(* Logix 5000 project; controller reports 1756-L63 rev 20.15; software revision 20.04; part 35 of 52 *)

        [32].log_data[44].total := -1012.85846, [32].log_data[44].time := 3600.0, [32].log_data[44].valid := 1, [32].log_data[45].time := 3600.0, [32].log_data[45].valid := 1, [32].log_data[46].time := 3600.0, [32].log_data[46].valid := 1, [32].log_data[47].time := 3600.0, [32].log_data[47].valid := 1, [32].log_data[48].min := 6.578031, [32].log_data[48].max := 6.9292355, [32].log_data[48].total := 24261.766, [32].log_data[48].time := 3600.0, [32].log_data[48].minminute := 9, [32].log_data[48].maxminute := 51, [32].log_data[48].valid := 1, [32].log_data[49].min := 7.0189543, [32].log_data[49].max := 9.474559, [32].log_data[49].total := 29951.562, [32].log_data[49].time := 3600.0, [32].log_data[49].minminute := 8, [32].log_data[49].maxminute := 45, [32].log_data[49].valid := 1, [32].log_data[50].min := 2.0610397, [32].log_data[50].max := 2.1768122, [32].log_data[50].total := 7588.2583, [32].log_data[50].time := 3600.0, [32].log_data[50].minminute := 44, [32].log_data[50].maxminute := 52, [32].log_data[50].valid := 1, [32].log_data[51].time := 3600.0, [32].log_data[51].valid := 1, [32].log_data[52].min := -3.0, [32].log_data[52].max := 0.13999939, [32].log_data[52].total := -7599.1304, [32].log_data[52].time := 3600.0, [32].log_data[52].minminute := 11, [32].log_data[52].valid := 1, [32].log_data[53].min := -2.5200043, [32].log_data[53].max := 0.17999268, [32].log_data[53].total := -6900.277, [32].log_data[53].time := 3600.0, [32].log_data[53].minminute := 27, [32].log_data[53].maxminute := 16, [32].log_data[53].valid := 1, [32].log_data[54].max := 0.554, [32].log_data[54].total := 1229.82, [32].log_data[54].time := 3600.0, [32].log_data[54].maxminute := 11, [32].log_data[54].valid := 1, [32].log_data[55].max := 0.523, [32].log_data[55].total := 1217.2505, [32].log_data[55].time := 3600.0, [32].log_data[55].minminute := 4, [32].log_data[55].maxminute := 58, [32].log_data[55].valid := 1, [32].log_data[56].min := 0.16024561, [32].log_data[56].max := 0.16067745, [32].log_data[56].total := 577.5993, [32].log_data[56].time := 3600.0,
        [32].log_data[56].minminute := 58, [32].log_data[56].maxminute := 2, [32].log_data[56].valid := 1, [32].log_data[57].min := 0.29596147, [32].log_data[57].max := 0.2979244, [32].log_data[57].total := 1067.1407, [32].log_data[57].time := 3600.0, [32].log_data[57].minminute := 25, [32].log_data[57].maxminute := 3, [32].log_data[57].valid := 1, [32].log_data[58].time := 3600.0, [32].log_data[58].valid := 1, [32].log_data[59].time := 3600.0, [32].log_data[59].valid := 1, [32].log_data[60].valid := 1, [32].log_data[61].valid := 1, [32].log_data[62].valid := 1, [32].log_data[63].valid := 1, [32].log_data[64].valid := 1, [32].log_data[65].valid := 1, [32].log_data[66].valid := 1, [32].log_data[67].valid := 1, [32].log_data[68].valid := 1, [32].log_data[69].valid := 1, [32].log_data[70].valid := 1, [32].log_data[71].valid := 1, [32].log_data[72].valid := 1, [32].log_data[73].valid := 1, [32].log_data[74].valid := 1, [32].log_data[75].valid := 1, [32].log_data[76].valid := 1, [32].log_data[77].valid := 1, [32].log_data[78].valid := 1, [32].log_data[79].valid := 1, [32].log_data[80].valid := 1, [32].log_data[81].valid := 1, [32].log_data[82].valid := 1, [32].log_data[83].valid := 1, [32].log_data[84].valid := 1, [32].log_data[85].valid := 1, [32].log_data[86].valid := 1, [32].log_data[87].valid := 1, [32].log_data[88].valid := 1, [32].log_data[89].valid := 1, [32].log_data[90].valid := 1, [32].log_data[91].valid := 1, [32].log_data[92].valid := 1, [32].log_data[93].valid := 1, [32].log_data[94].valid := 1, [32].log_data[95].valid := 1, [32].log_data[96].valid := 1, [32].log_data[97].valid := 1, [32].log_data[98].valid := 1, [32].log_data[99].valid := 1, [32].log_data[100].valid := 1, [32].log_data[101].valid := 1, [32].log_data[102].valid := 1, [32].log_data[103].valid := 1, [32].log_data[104].valid := 1, [32].log_data[105].valid := 1,
        [32].log_data[106].valid := 1, [32].log_data[107].valid := 1, [32].log_data[108].valid := 1, [32].log_data[109].valid := 1, [32].log_data[110].valid := 1, [32].log_data[111].valid := 1, [32].log_data[112].valid := 1, [32].log_data[113].valid := 1, [32].log_data[114].valid := 1, [32].log_data[115].valid := 1, [32].log_data[116].valid := 1, [32].log_data[117].valid := 1, [32].log_data[118].valid := 1, [32].log_data[119].valid := 1, [32].log_data[120].valid := 1, [32].log_data[121].valid := 1, [32].log_data[122].valid := 1, [32].log_data[123].valid := 1, [32].log_data[124].valid := 1, [32].time.Year := 2023, [32].time.Month := 1, [32].time.Day := 14, [32].time.Hour := 11, [32].time.Minute := 59, [32].time.Second := 59, [33].log_data[0].min := 1.0, [33].log_data[0].max := 1.0, [33].log_data[0].total := 3599.5, [33].log_data[0].time := 3599.5, [33].log_data[0].valid := 1, [33].log_data[1].time := 3599.5, [33].log_data[1].valid := 1, [33].log_data[2].time := 3599.5, [33].log_data[2].valid := 1, [33].log_data[3].time := 3599.5, [33].log_data[3].valid := 1, [33].log_data[4].time := 3599.5, [33].log_data[4].valid := 1, [33].log_data[5].time := 3599.5, [33].log_data[5].valid := 1, [33].log_data[6].time := 3599.5, [33].log_data[6].valid := 1, [33].log_data[7].time := 3599.5, [33].log_data[7].valid := 1, [33].log_data[8].min := 1.0, [33].log_data[8].max := 1.0, [33].log_data[8].total := 3599.5, [33].log_data[8].time := 3599.5, [33].log_data[8].valid := 1, [33].log_data[9].min := 1.0, [33].log_data[9].max := 1.0, [33].log_data[9].total := 3599.5, [33].log_data[9].time := 3599.5, [33].log_data[9].valid := 1, [33].log_data[10].min := 1.0, [33].log_data[10].max := 1.0, [33].log_data[10].total := 3599.5, [33].log_data[10].time := 3599.5, [33].log_data[10].valid := 1, [33].log_data[11].time := 3599.5,
        [33].log_data[11].valid := 1, [33].log_data[12].min := 1.0, [33].log_data[12].max := 1.0, [33].log_data[12].total := 3599.5, [33].log_data[12].time := 3599.5, [33].log_data[12].valid := 1, [33].log_data[13].min := 1.0, [33].log_data[13].max := 1.0, [33].log_data[13].total := 3599.5, [33].log_data[13].time := 3599.5, [33].log_data[13].valid := 1, [33].log_data[14].time := 3599.5, [33].log_data[14].valid := 1, [33].log_data[15].time := 3599.5, [33].log_data[15].valid := 1, [33].log_data[16].time := 3599.5, [33].log_data[16].valid := 1, [33].log_data[17].min := 1.0, [33].log_data[17].max := 1.0, [33].log_data[17].total := 3599.5, [33].log_data[17].time := 3599.5, [33].log_data[17].valid := 1, [33].log_data[18].time := 3599.5, [33].log_data[18].valid := 1, [33].log_data[19].time := 3599.5, [33].log_data[19].valid := 1, [33].log_data[20].time := 3599.5, [33].log_data[20].valid := 1, [33].log_data[21].min := 1.0, [33].log_data[21].max := 1.0, [33].log_data[21].total := 3599.5, [33].log_data[21].time := 3599.5, [33].log_data[21].valid := 1, [33].log_data[22].time := 3599.5, [33].log_data[22].valid := 1, [33].log_data[23].time := 3599.5, [33].log_data[23].valid := 1, [33].log_data[24].time := 3599.5, [33].log_data[24].valid := 1, [33].log_data[25].time := 3599.5, [33].log_data[25].valid := 1, [33].log_data[26].time := 3599.5, [33].log_data[26].valid := 1, [33].log_data[27].time := 3599.5, [33].log_data[27].valid := 1, [33].log_data[28].time := 3599.5, [33].log_data[28].valid := 1, [33].log_data[29].min := 1.0, [33].log_data[29].max := 1.0, [33].log_data[29].total := 3599.5, [33].log_data[29].time := 3599.5, [33].log_data[29].valid := 1, [33].log_data[30].min := 1.0, [33].log_data[30].max := 1.0, [33].log_data[30].total := 3599.5, [33].log_data[30].time := 3599.5, [33].log_data[30].valid := 1, [33].log_data[31].max := 1.0, [33].log_data[31].total := 1440.498, [33].log_data[31].time := 3599.5,
        [33].log_data[31].minminute := 2, [33].log_data[31].valid := 1, [33].log_data[32].max := 1.0, [33].log_data[32].total := 1629.7471, [33].log_data[32].time := 3599.5, [33].log_data[32].maxminute := 4, [33].log_data[32].valid := 1, [33].log_data[33].time := 3599.5, [33].log_data[33].valid := 1, [33].log_data[34].time := 3599.5, [33].log_data[34].valid := 1, [33].log_data[35].max := 1.0, [33].log_data[35].total := 1618.7471, [33].log_data[35].time := 3599.5, [33].log_data[35].maxminute := 9, [33].log_data[35].valid := 1, [33].log_data[36].max := 1.0, [33].log_data[36].total := 1539.498, [33].log_data[36].time := 3599.5, [33].log_data[36].minminute := 7, [33].log_data[36].valid := 1, [33].log_data[37].time := 3599.5, [33].log_data[37].valid := 1, [33].log_data[38].time := 3599.5, [33].log_data[38].valid := 1, [33].log_data[39].min := 1.0018904, [33].log_data[39].max := 1.0133146, [33].log_data[39].total := 3629.6885, [33].log_data[39].time := 3599.5, [33].log_data[39].minminute := 3, [33].log_data[39].maxminute := 54, [33].log_data[39].valid := 1, [33].log_data[40].min := 7.54453, [33].log_data[40].max := 7.597843, [33].log_data[40].total := 27288.283, [33].log_data[40].time := 3599.5, [33].log_data[40].minminute := 36, [33].log_data[40].maxminute := 39, [33].log_data[40].valid := 1, [33].log_data[41].min := 0.03392505, [33].log_data[41].max := 0.0455061, [33].log_data[41].total := 141.35881, [33].log_data[41].time := 3599.5, [33].log_data[41].minminute := 21, [33].log_data[41].maxminute := 14, [33].log_data[41].valid := 1, [33].log_data[42].min := 2.2922316, [33].log_data[42].max := 2.297178, [33].log_data[42].total := 8261.017, [33].log_data[42].time := 3599.5, [33].log_data[42].minminute := 53, [33].log_data[42].maxminute := 2, [33].log_data[42].valid := 1, [33].log_data[43].min := -0.26000214, [33].log_data[43].max := -0.26000214, [33].log_data[43].total := -935.8432, [33].log_data[43].time := 3599.5, [33].log_data[43].valid := 1, [33].log_data[44].min := -0.30000305, [33].log_data[44].max := -0.27999878,
        [33].log_data[44].total := -1048.7408, [33].log_data[44].time := 3599.5, [33].log_data[44].valid := 1, [33].log_data[45].time := 3599.5, [33].log_data[45].valid := 1, [33].log_data[46].time := 3599.5, [33].log_data[46].valid := 1, [33].log_data[47].time := 3599.5, [33].log_data[47].valid := 1, [33].log_data[48].min := 6.5807796, [33].log_data[48].max := 6.786885, [33].log_data[48].total := 24167.266, [33].log_data[48].time := 3599.5, [33].log_data[48].minminute := 15, [33].log_data[48].maxminute := 30, [33].log_data[48].valid := 1, [33].log_data[49].min := 7.0046253, [33].log_data[49].max := 9.562302, [33].log_data[49].total := 29994.54, [33].log_data[49].time := 3599.5, [33].log_data[49].minminute := 12, [33].log_data[49].maxminute := 58, [33].log_data[49].valid := 1, [33].log_data[50].min := 2.0844767, [33].log_data[50].max := 2.1683326, [33].log_data[50].total := 7656.986, [33].log_data[50].time := 3599.5, [33].log_data[50].minminute := 59, [33].log_data[50].valid := 1, [33].log_data[51].time := 3599.5, [33].log_data[51].valid := 1, [33].log_data[52].min := -3.040001, [33].log_data[52].max := 0.13999939, [33].log_data[52].total := -7548.99, [33].log_data[52].time := 3599.5, [33].log_data[52].minminute := 56, [33].log_data[52].maxminute := 3, [33].log_data[52].valid := 1, [33].log_data[53].min := -2.4800034, [33].log_data[53].max := 0.22000122, [33].log_data[53].total := -7164.744, [33].log_data[53].time := 3599.5, [33].log_data[53].minminute := 9, [33].log_data[53].maxminute := 9, [33].log_data[53].valid := 1, [33].log_data[54].max := 0.5475, [33].log_data[54].total := 1216.9542, [33].log_data[54].time := 3599.5, [33].log_data[54].minminute := 2, [33].log_data[54].maxminute := 56, [33].log_data[54].valid := 1, [33].log_data[55].max := 0.5295, [33].log_data[55].total := 1254.2496, [33].log_data[55].time := 3599.5, [33].log_data[55].minminute := 7, [33].log_data[55].maxminute := 51, [33].log_data[55].valid := 1, [33].log_data[56].min := 0.16024561, [33].log_data[56].max := 0.16063818, [33].log_data[56].total := 577.4036,
        [33].log_data[56].time := 3599.5, [33].log_data[56].minminute := 9, [33].log_data[56].maxminute := 1, [33].log_data[56].valid := 1, [33].log_data[57].min := 0.29446968, [33].log_data[57].max := 0.29627553, [33].log_data[57].total := 1062.121, [33].log_data[57].time := 3599.5, [33].log_data[57].minminute := 54, [33].log_data[57].maxminute := 1, [33].log_data[57].valid := 1, [33].log_data[58].time := 3599.5, [33].log_data[58].valid := 1, [33].log_data[59].time := 3599.5, [33].log_data[59].valid := 1, [33].log_data[60].valid := 1, [33].log_data[61].valid := 1, [33].log_data[62].valid := 1, [33].log_data[63].valid := 1, [33].log_data[64].valid := 1, [33].log_data[65].valid := 1, [33].log_data[66].valid := 1, [33].log_data[67].valid := 1, [33].log_data[68].valid := 1, [33].log_data[69].valid := 1, [33].log_data[70].valid := 1, [33].log_data[71].valid := 1, [33].log_data[72].valid := 1, [33].log_data[73].valid := 1, [33].log_data[74].valid := 1, [33].log_data[75].valid := 1, [33].log_data[76].valid := 1, [33].log_data[77].valid := 1, [33].log_data[78].valid := 1, [33].log_data[79].valid := 1, [33].log_data[80].valid := 1, [33].log_data[81].valid := 1, [33].log_data[82].valid := 1, [33].log_data[83].valid := 1, [33].log_data[84].valid := 1, [33].log_data[85].valid := 1, [33].log_data[86].valid := 1, [33].log_data[87].valid := 1, [33].log_data[88].valid := 1, [33].log_data[89].valid := 1, [33].log_data[90].valid := 1, [33].log_data[91].valid := 1, [33].log_data[92].valid := 1, [33].log_data[93].valid := 1, [33].log_data[94].valid := 1, [33].log_data[95].valid := 1, [33].log_data[96].valid := 1, [33].log_data[97].valid := 1, [33].log_data[98].valid := 1, [33].log_data[99].valid := 1, [33].log_data[100].valid := 1, [33].log_data[101].valid := 1, [33].log_data[102].valid := 1, [33].log_data[103].valid := 1, [33].log_data[104].valid := 1,
        [33].log_data[105].valid := 1, [33].log_data[106].valid := 1, [33].log_data[107].valid := 1, [33].log_data[108].valid := 1, [33].log_data[109].valid := 1, [33].log_data[110].valid := 1, [33].log_data[111].valid := 1, [33].log_data[112].valid := 1, [33].log_data[113].valid := 1, [33].log_data[114].valid := 1, [33].log_data[115].valid := 1, [33].log_data[116].valid := 1, [33].log_data[117].valid := 1, [33].log_data[118].valid := 1, [33].log_data[119].valid := 1, [33].log_data[120].valid := 1, [33].log_data[121].valid := 1, [33].log_data[122].valid := 1, [33].log_data[123].valid := 1, [33].log_data[124].valid := 1, [33].time.Year := 2023, [33].time.Month := 1, [33].time.Day := 14, [33].time.Hour := 12, [33].time.Minute := 59, [33].time.Second := 59, [34].log_data[0].min := 1.0, [34].log_data[0].max := 1.0, [34].log_data[0].total := 3600.0, [34].log_data[0].time := 3600.0, [34].log_data[0].valid := 1, [34].log_data[1].max := 1.0, [34].log_data[1].total := 563.0, [34].log_data[1].time := 3600.0, [34].log_data[1].maxminute := 16, [34].log_data[1].valid := 1, [34].log_data[2].max := 1.0, [34].log_data[2].total := 559.5, [34].log_data[2].time := 3600.0, [34].log_data[2].maxminute := 16, [34].log_data[2].valid := 1, [34].log_data[3].time := 3600.0, [34].log_data[3].valid := 1, [34].log_data[4].time := 3600.0, [34].log_data[4].valid := 1, [34].log_data[5].max := 1.0, [34].log_data[5].total := 265.5, [34].log_data[5].time := 3600.0, [34].log_data[5].maxminute := 18, [34].log_data[5].valid := 1, [34].log_data[6].time := 3600.0, [34].log_data[6].valid := 1, [34].log_data[7].time := 3600.0, [34].log_data[7].valid := 1, [34].log_data[8].min := 1.0, [34].log_data[8].max := 1.0, [34].log_data[8].total := 3600.0, [34].log_data[8].time := 3600.0, [34].log_data[8].valid := 1, [34].log_data[9].min := 1.0,
        [34].log_data[9].max := 1.0, [34].log_data[9].total := 3600.0, [34].log_data[9].time := 3600.0, [34].log_data[9].valid := 1, [34].log_data[10].min := 1.0, [34].log_data[10].max := 1.0, [34].log_data[10].total := 3600.0, [34].log_data[10].time := 3600.0, [34].log_data[10].valid := 1, [34].log_data[11].time := 3600.0, [34].log_data[11].valid := 1, [34].log_data[12].min := 1.0, [34].log_data[12].max := 1.0, [34].log_data[12].total := 3600.0, [34].log_data[12].time := 3600.0, [34].log_data[12].valid := 1, [34].log_data[13].min := 1.0, [34].log_data[13].max := 1.0, [34].log_data[13].total := 3600.0, [34].log_data[13].time := 3600.0, [34].log_data[13].valid := 1, [34].log_data[14].time := 3600.0, [34].log_data[14].valid := 1, [34].log_data[15].time := 3600.0, [34].log_data[15].valid := 1, [34].log_data[16].time := 3600.0, [34].log_data[16].valid := 1, [34].log_data[17].min := 1.0, [34].log_data[17].max := 1.0, [34].log_data[17].total := 3600.0, [34].log_data[17].time := 3600.0, [34].log_data[17].valid := 1, [34].log_data[18].time := 3600.0, [34].log_data[18].valid := 1, [34].log_data[19].time := 3600.0, [34].log_data[19].valid := 1, [34].log_data[20].time := 3600.0, [34].log_data[20].valid := 1, [34].log_data[21].min := 1.0, [34].log_data[21].max := 1.0, [34].log_data[21].total := 3600.0, [34].log_data[21].time := 3600.0, [34].log_data[21].valid := 1, [34].log_data[22].time := 3600.0, [34].log_data[22].valid := 1, [34].log_data[23].time := 3600.0, [34].log_data[23].valid := 1, [34].log_data[24].time := 3600.0, [34].log_data[24].valid := 1, [34].log_data[25].time := 3600.0, [34].log_data[25].valid := 1, [34].log_data[26].time := 3600.0, [34].log_data[26].valid := 1, [34].log_data[27].time := 3600.0, [34].log_data[27].valid := 1, [34].log_data[28].time := 3600.0, [34].log_data[28].valid := 1, [34].log_data[29].min := 1.0, [34].log_data[29].max := 1.0, [34].log_data[29].total := 3600.0,
        [34].log_data[29].time := 3600.0, [34].log_data[29].valid := 1, [34].log_data[30].min := 1.0, [34].log_data[30].max := 1.0, [34].log_data[30].total := 3600.0, [34].log_data[30].time := 3600.0, [34].log_data[30].valid := 1, [34].log_data[31].max := 1.0, [34].log_data[31].total := 1440.998, [34].log_data[31].time := 3600.0, [34].log_data[31].minminute := 5, [34].log_data[31].valid := 1, [34].log_data[32].max := 1.0, [34].log_data[32].total := 1630.249, [34].log_data[32].time := 3600.0, [34].log_data[32].maxminute := 7, [34].log_data[32].valid := 1, [34].log_data[33].time := 3600.0, [34].log_data[33].valid := 1, [34].log_data[34].time := 3600.0, [34].log_data[34].valid := 1, [34].log_data[35].max := 1.0, [34].log_data[35].total := 1440.7471, [34].log_data[35].time := 3600.0, [34].log_data[35].valid := 1, [34].log_data[36].max := 1.0, [34].log_data[36].total := 1629.7471, [34].log_data[36].time := 3600.0, [34].log_data[36].maxminute := 1, [34].log_data[36].valid := 1, [34].log_data[37].max := 7.2674255, [34].log_data[37].total := 3545.5764, [34].log_data[37].time := 3600.0, [34].log_data[37].maxminute := 17, [34].log_data[37].valid := 1, [34].log_data[38].time := 3600.0, [34].log_data[38].valid := 1, [34].log_data[39].min := 0.99541295, [34].log_data[39].max := 1.0230899, [34].log_data[39].total := 3616.9822, [34].log_data[39].time := 3600.0, [34].log_data[39].minminute := 53, [34].log_data[39].maxminute := 23, [34].log_data[39].valid := 1, [34].log_data[40].min := 7.5659657, [34].log_data[40].max := 7.597568, [34].log_data[40].total := 27297.441, [34].log_data[40].time := 3600.0, [34].log_data[40].minminute := 4, [34].log_data[40].valid := 1, [34].log_data[41].min := 0.026858643, [34].log_data[41].max := 0.04040259, [34].log_data[41].total := 123.13823, [34].log_data[41].time := 3600.0, [34].log_data[41].minminute := 46, [34].log_data[41].maxminute := 20, [34].log_data[41].valid := 1, [34].log_data[42].min := 2.2921138, [34].log_data[42].max := 2.297296, [34].log_data[42].total := 8262.21,
        [34].log_data[42].time := 3600.0, [34].log_data[42].minminute := 16, [34].log_data[42].maxminute := 19, [34].log_data[42].valid := 1, [34].log_data[43].min := -0.27999878, [34].log_data[43].max := -0.26000214, [34].log_data[43].total := -936.07263, [34].log_data[43].time := 3600.0, [34].log_data[43].minminute := 42, [34].log_data[43].valid := 1, [34].log_data[44].min := -0.30000305, [34].log_data[44].max := -0.27999878, [34].log_data[44].total := -1079.2913, [34].log_data[44].time := 3600.0, [34].log_data[44].valid := 1, [34].log_data[45].time := 3600.0, [34].log_data[45].valid := 1, [34].log_data[46].time := 3600.0, [34].log_data[46].valid := 1, [34].log_data[47].time := 3600.0, [34].log_data[47].valid := 1, [34].log_data[48].min := 6.5807796, [34].log_data[48].max := 6.9448996, [34].log_data[48].total := 24212.871, [34].log_data[48].time := 3600.0, [34].log_data[48].minminute := 50, [34].log_data[48].maxminute := 25, [34].log_data[48].valid := 1, [34].log_data[49].min := 6.9066753, [34].log_data[49].max := 9.627471, [34].log_data[49].total := 29711.473, [34].log_data[49].time := 3600.0, [34].log_data[49].minminute := 48, [34].log_data[49].maxminute := 18, [34].log_data[49].valid := 1, [34].log_data[50].min := 2.0580952, [34].log_data[50].max := 2.1809344, [34].log_data[50].total := 7661.901, [34].log_data[50].time := 3600.0, [34].log_data[50].minminute := 17, [34].log_data[50].maxminute := 28, [34].log_data[50].valid := 1, [34].log_data[51].time := 3600.0, [34].log_data[51].valid := 1, [34].log_data[52].min := -2.9400024, [34].log_data[52].max := 0.11999512, [34].log_data[52].total := -7502.3184, [34].log_data[52].time := 3600.0, [34].log_data[52].minminute := 59, [34].log_data[52].maxminute := 5, [34].log_data[52].valid := 1, [34].log_data[53].min := -2.4800034, [34].log_data[53].max := 0.22000122, [34].log_data[53].total := -6940.3506, [34].log_data[53].time := 3600.0, [34].log_data[53].minminute := 8, [34].log_data[53].maxminute := 1, [34].log_data[53].valid := 1, [34].log_data[54].max := 0.5335, [34].log_data[54].total := 1218.3517,
        [34].log_data[54].time := 3600.0, [34].log_data[54].minminute := 5, [34].log_data[54].maxminute := 7, [34].log_data[54].valid := 1, [34].log_data[55].max := 0.51600003, [34].log_data[55].total := 1216.9606, [34].log_data[55].time := 3600.0, [34].log_data[55].maxminute := 12, [34].log_data[55].valid := 1, [34].log_data[56].min := 0.16012783, [34].log_data[56].max := 0.16067745, [34].log_data[56].total := 577.3217, [34].log_data[56].time := 3600.0, [34].log_data[56].minminute := 17, [34].log_data[56].maxminute := 2, [34].log_data[56].valid := 1, [34].log_data[57].min := 0.29286006, [34].log_data[57].max := 0.29490152, [34].log_data[57].total := 1059.95, [34].log_data[57].time := 3600.0, [34].log_data[57].minminute := 58, [34].log_data[57].maxminute := 1, [34].log_data[57].valid := 1, [34].log_data[58].time := 3600.0, [34].log_data[58].valid := 1, [34].log_data[59].time := 3600.0, [34].log_data[59].valid := 1, [34].log_data[60].valid := 1, [34].log_data[61].valid := 1, [34].log_data[62].valid := 1, [34].log_data[63].valid := 1, [34].log_data[64].valid := 1, [34].log_data[65].valid := 1, [34].log_data[66].valid := 1, [34].log_data[67].valid := 1, [34].log_data[68].valid := 1, [34].log_data[69].valid := 1, [34].log_data[70].valid := 1, [34].log_data[71].valid := 1, [34].log_data[72].valid := 1, [34].log_data[73].valid := 1, [34].log_data[74].valid := 1, [34].log_data[75].valid := 1, [34].log_data[76].valid := 1, [34].log_data[77].valid := 1, [34].log_data[78].valid := 1, [34].log_data[79].valid := 1, [34].log_data[80].valid := 1, [34].log_data[81].valid := 1, [34].log_data[82].valid := 1, [34].log_data[83].valid := 1, [34].log_data[84].valid := 1, [34].log_data[85].valid := 1, [34].log_data[86].valid := 1, [34].log_data[87].valid := 1, [34].log_data[88].valid := 1, [34].log_data[89].valid := 1, [34].log_data[90].valid := 1, [34].log_data[91].valid := 1, [34].log_data[92].valid := 1,
        [34].log_data[93].valid := 1, [34].log_data[94].valid := 1, [34].log_data[95].valid := 1, [34].log_data[96].valid := 1, [34].log_data[97].valid := 1, [34].log_data[98].valid := 1, [34].log_data[99].valid := 1, [34].log_data[100].valid := 1, [34].log_data[101].valid := 1, [34].log_data[102].valid := 1, [34].log_data[103].valid := 1, [34].log_data[104].valid := 1, [34].log_data[105].valid := 1, [34].log_data[106].valid := 1, [34].log_data[107].valid := 1, [34].log_data[108].valid := 1, [34].log_data[109].valid := 1, [34].log_data[110].valid := 1, [34].log_data[111].valid := 1, [34].log_data[112].valid := 1, [34].log_data[113].valid := 1, [34].log_data[114].valid := 1, [34].log_data[115].valid := 1, [34].log_data[116].valid := 1, [34].log_data[117].valid := 1, [34].log_data[118].valid := 1, [34].log_data[119].valid := 1, [34].log_data[120].valid := 1, [34].log_data[121].valid := 1, [34].log_data[122].valid := 1, [34].log_data[123].valid := 1, [34].log_data[124].valid := 1, [34].time.Year := 2023, [34].time.Month := 1, [34].time.Day := 14, [34].time.Hour := 13, [34].time.Minute := 59, [34].time.Second := 59, [35].log_data[0].min := 1.0, [35].log_data[0].max := 1.0, [35].log_data[0].total := 3600.0, [35].log_data[0].time := 3600.0, [35].log_data[0].valid := 1, [35].log_data[1].max := 1.0, [35].log_data[1].total := 532.0, [35].log_data[1].time := 3600.0, [35].log_data[1].maxminute := 41, [35].log_data[1].valid := 1, [35].log_data[2].max := 1.0, [35].log_data[2].total := 528.5, [35].log_data[2].time := 3600.0, [35].log_data[2].maxminute := 41, [35].log_data[2].valid := 1, [35].log_data[3].time := 3600.0, [35].log_data[3].valid := 1, [35].log_data[4].time := 3600.0, [35].log_data[4].valid := 1, [35].log_data[5].max := 1.0, [35].log_data[5].total := 237.0, [35].log_data[5].time := 3600.0,
        [35].log_data[5].maxminute := 43, [35].log_data[5].valid := 1, [35].log_data[6].time := 3600.0, [35].log_data[6].valid := 1, [35].log_data[7].time := 3600.0, [35].log_data[7].valid := 1, [35].log_data[8].min := 1.0, [35].log_data[8].max := 1.0, [35].log_data[8].total := 3600.0, [35].log_data[8].time := 3600.0, [35].log_data[8].valid := 1, [35].log_data[9].min := 1.0, [35].log_data[9].max := 1.0, [35].log_data[9].total := 3600.0, [35].log_data[9].time := 3600.0, [35].log_data[9].valid := 1, [35].log_data[10].min := 1.0, [35].log_data[10].max := 1.0, [35].log_data[10].total := 3600.0, [35].log_data[10].time := 3600.0, [35].log_data[10].valid := 1, [35].log_data[11].time := 3600.0, [35].log_data[11].valid := 1, [35].log_data[12].min := 1.0, [35].log_data[12].max := 1.0, [35].log_data[12].total := 3600.0, [35].log_data[12].time := 3600.0, [35].log_data[12].valid := 1, [35].log_data[13].min := 1.0, [35].log_data[13].max := 1.0, [35].log_data[13].total := 3600.0, [35].log_data[13].time := 3600.0, [35].log_data[13].valid := 1, [35].log_data[14].time := 3600.0, [35].log_data[14].valid := 1, [35].log_data[15].time := 3600.0, [35].log_data[15].valid := 1, [35].log_data[16].time := 3600.0, [35].log_data[16].valid := 1, [35].log_data[17].min := 1.0, [35].log_data[17].max := 1.0, [35].log_data[17].total := 3600.0, [35].log_data[17].time := 3600.0, [35].log_data[17].valid := 1, [35].log_data[18].time := 3600.0, [35].log_data[18].valid := 1, [35].log_data[19].time := 3600.0, [35].log_data[19].valid := 1, [35].log_data[20].time := 3600.0, [35].log_data[20].valid := 1, [35].log_data[21].min := 1.0, [35].log_data[21].max := 1.0, [35].log_data[21].total := 3600.0, [35].log_data[21].time := 3600.0, [35].log_data[21].valid := 1, [35].log_data[22].time := 3600.0, [35].log_data[22].valid := 1, [35].log_data[23].time := 3600.0, [35].log_data[23].valid := 1, [35].log_data[24].time := 3600.0,
        [35].log_data[24].valid := 1, [35].log_data[25].time := 3600.0, [35].log_data[25].valid := 1, [35].log_data[26].time := 3600.0, [35].log_data[26].valid := 1, [35].log_data[27].time := 3600.0, [35].log_data[27].valid := 1, [35].log_data[28].time := 3600.0, [35].log_data[28].valid := 1, [35].log_data[29].min := 1.0, [35].log_data[29].max := 1.0, [35].log_data[29].total := 3600.0, [35].log_data[29].time := 3600.0, [35].log_data[29].valid := 1, [35].log_data[30].min := 1.0, [35].log_data[30].max := 1.0, [35].log_data[30].total := 3600.0, [35].log_data[30].time := 3600.0, [35].log_data[30].valid := 1, [35].log_data[31].max := 1.0, [35].log_data[31].total := 1620.749, [35].log_data[31].time := 3600.0, [35].log_data[31].minminute := 8, [35].log_data[31].valid := 1, [35].log_data[32].max := 1.0, [35].log_data[32].total := 1538.2471, [35].log_data[32].time := 3600.0, [35].log_data[32].maxminute := 10, [35].log_data[32].valid := 1, [35].log_data[33].time := 3600.0, [35].log_data[33].valid := 1, [35].log_data[34].time := 3600.0, [35].log_data[34].valid := 1, [35].log_data[35].max := 1.0, [35].log_data[35].total := 1440.7471, [35].log_data[35].time := 3600.0, [35].log_data[35].minminute := 3, [35].log_data[35].valid := 1, [35].log_data[36].max := 1.0, [35].log_data[36].total := 1629.7471, [35].log_data[36].time := 3600.0, [35].log_data[36].maxminute := 4, [35].log_data[36].valid := 1, [35].log_data[37].max := 7.5944467, [35].log_data[37].total := 3511.0564, [35].log_data[37].time := 3600.0, [35].log_data[37].maxminute := 42, [35].log_data[37].valid := 1, [35].log_data[38].time := 3600.0, [35].log_data[38].valid := 1, [35].log_data[39].min := 0.995884, [35].log_data[39].max := 1.0227365, [35].log_data[39].total := 3610.0178, [35].log_data[39].time := 3600.0, [35].log_data[39].minminute := 14, [35].log_data[39].maxminute := 48, [35].log_data[39].valid := 1, [35].log_data[40].min := 7.551675, [35].log_data[40].max := 7.600591, [35].log_data[40].total := 27302.318,
        [35].log_data[40].time := 3600.0, [35].log_data[40].minminute := 6, [35].log_data[40].maxminute := 9, [35].log_data[40].valid := 1, [35].log_data[41].min := 0.027054932, [35].log_data[41].max := 0.053750485, [35].log_data[41].total := 143.93544, [35].log_data[41].time := 3600.0, [35].log_data[41].minminute := 13, [35].log_data[41].maxminute := 24, [35].log_data[41].valid := 1, [35].log_data[42].min := 2.292467, [35].log_data[42].max := 2.297178, [35].log_data[42].total := 8262.258, [35].log_data[42].time := 3600.0, [35].log_data[42].minminute := 11, [35].log_data[42].valid := 1, [35].log_data[43].min := -0.27999878, [35].log_data[43].max := -0.26000214, [35].log_data[43].total := -937.09906, [35].log_data[43].time := 3600.0, [35].log_data[43].valid := 1, [35].log_data[44].min := -0.30000305, [35].log_data[44].max := -0.27999878, [35].log_data[44].total := -1080.081, [35].log_data[44].time := 3600.0, [35].log_data[44].maxminute := 11, [35].log_data[44].valid := 1, [35].log_data[45].time := 3600.0, [35].log_data[45].valid := 1, [35].log_data[46].time := 3600.0, [35].log_data[46].valid := 1, [35].log_data[47].time := 3600.0, [35].log_data[47].valid := 1, [35].log_data[48].min := 6.69455, [35].log_data[48].max := 6.9534187, [35].log_data[48].total := 24376.504, [35].log_data[48].time := 3600.0, [35].log_data[48].minminute := 59, [35].log_data[48].maxminute := 46, [35].log_data[48].valid := 1, [35].log_data[49].min := 7.375222, [35].log_data[49].max := 9.60313, [35].log_data[49].total := 32263.094, [35].log_data[49].time := 3600.0, [35].log_data[49].minminute := 59, [35].log_data[49].maxminute := 43, [35].log_data[49].valid := 1, [35].log_data[50].min := 2.0739946, [35].log_data[50].max := 2.1845853, [35].log_data[50].total := 7637.917, [35].log_data[50].time := 3600.0, [35].log_data[50].minminute := 43, [35].log_data[50].maxminute := 50, [35].log_data[50].valid := 1, [35].log_data[51].time := 3600.0, [35].log_data[51].valid := 1, [35].log_data[52].min := -2.7799988, [35].log_data[52].max := 0.11999512, [35].log_data[52].total := -7737.476,
        [35].log_data[52].time := 3600.0, [35].log_data[52].minminute := 31, [35].log_data[52].maxminute := 8, [35].log_data[52].valid := 1, [35].log_data[53].min := -2.6399994, [35].log_data[53].max := 0.22000122, [35].log_data[53].total := -6976.84, [35].log_data[53].time := 3600.0, [35].log_data[53].minminute := 4, [35].log_data[53].maxminute := 4, [35].log_data[53].valid := 1, [35].log_data[54].max := 0.5385, [35].log_data[54].total := 1253.9543, [35].log_data[54].time := 3600.0, [35].log_data[54].minminute := 8, [35].log_data[54].maxminute := 31, [35].log_data[54].valid := 1, [35].log_data[55].max := 0.5305, [35].log_data[55].total := 1217.441, [35].log_data[55].time := 3600.0, [35].log_data[55].minminute := 3, [35].log_data[55].maxminute := 4, [35].log_data[55].valid := 1, [35].log_data[56].min := 0.16012783, [35].log_data[56].max := 0.16055967, [35].log_data[56].total := 577.202, [35].log_data[56].time := 3600.0, [35].log_data[56].maxminute := 4, [35].log_data[56].valid := 1, [35].log_data[57].min := 0.29278153, [35].log_data[57].max := 0.29321337, [35].log_data[57].total := 1054.7292, [35].log_data[57].time := 3600.0, [35].log_data[57].minminute := 35, [35].log_data[57].maxminute := 2, [35].log_data[57].valid := 1, [35].log_data[58].time := 3600.0, [35].log_data[58].valid := 1, [35].log_data[59].time := 3600.0, [35].log_data[59].valid := 1, [35].log_data[60].valid := 1, [35].log_data[61].valid := 1, [35].log_data[62].valid := 1, [35].log_data[63].valid := 1, [35].log_data[64].valid := 1, [35].log_data[65].valid := 1, [35].log_data[66].valid := 1, [35].log_data[67].valid := 1, [35].log_data[68].valid := 1, [35].log_data[69].valid := 1, [35].log_data[70].valid := 1, [35].log_data[71].valid := 1, [35].log_data[72].valid := 1, [35].log_data[73].valid := 1, [35].log_data[74].valid := 1, [35].log_data[75].valid := 1, [35].log_data[76].valid := 1, [35].log_data[77].valid := 1, [35].log_data[78].valid := 1, [35].log_data[79].valid := 1,
        [35].log_data[80].valid := 1, [35].log_data[81].valid := 1, [35].log_data[82].valid := 1, [35].log_data[83].valid := 1, [35].log_data[84].valid := 1, [35].log_data[85].valid := 1, [35].log_data[86].valid := 1, [35].log_data[87].valid := 1, [35].log_data[88].valid := 1, [35].log_data[89].valid := 1, [35].log_data[90].valid := 1, [35].log_data[91].valid := 1, [35].log_data[92].valid := 1, [35].log_data[93].valid := 1, [35].log_data[94].valid := 1, [35].log_data[95].valid := 1, [35].log_data[96].valid := 1, [35].log_data[97].valid := 1, [35].log_data[98].valid := 1, [35].log_data[99].valid := 1, [35].log_data[100].valid := 1, [35].log_data[101].valid := 1, [35].log_data[102].valid := 1, [35].log_data[103].valid := 1, [35].log_data[104].valid := 1, [35].log_data[105].valid := 1, [35].log_data[106].valid := 1, [35].log_data[107].valid := 1, [35].log_data[108].valid := 1, [35].log_data[109].valid := 1, [35].log_data[110].valid := 1, [35].log_data[111].valid := 1, [35].log_data[112].valid := 1, [35].log_data[113].valid := 1, [35].log_data[114].valid := 1, [35].log_data[115].valid := 1, [35].log_data[116].valid := 1, [35].log_data[117].valid := 1, [35].log_data[118].valid := 1, [35].log_data[119].valid := 1, [35].log_data[120].valid := 1, [35].log_data[121].valid := 1, [35].log_data[122].valid := 1, [35].log_data[123].valid := 1, [35].log_data[124].valid := 1, [35].time.Year := 2023, [35].time.Month := 1, [35].time.Day := 14, [35].time.Hour := 14, [35].time.Minute := 59, [35].time.Second := 59, [36].log_data[0].min := 1.0, [36].log_data[0].max := 1.0, [36].log_data[0].total := 3600.0, [36].log_data[0].time := 3600.0, [36].log_data[0].valid := 1, [36].log_data[1].time := 3600.0, [36].log_data[1].valid := 1, [36].log_data[2].time := 3600.0, [36].log_data[2].valid := 1,
        [36].log_data[3].time := 3600.0, [36].log_data[3].valid := 1, [36].log_data[4].time := 3600.0, [36].log_data[4].valid := 1, [36].log_data[5].time := 3600.0, [36].log_data[5].valid := 1, [36].log_data[6].time := 3600.0, [36].log_data[6].valid := 1, [36].log_data[7].time := 3600.0, [36].log_data[7].valid := 1, [36].log_data[8].min := 1.0, [36].log_data[8].max := 1.0, [36].log_data[8].total := 3600.0, [36].log_data[8].time := 3600.0, [36].log_data[8].valid := 1, [36].log_data[9].min := 1.0, [36].log_data[9].max := 1.0, [36].log_data[9].total := 3600.0, [36].log_data[9].time := 3600.0, [36].log_data[9].valid := 1, [36].log_data[10].min := 1.0, [36].log_data[10].max := 1.0, [36].log_data[10].total := 3600.0, [36].log_data[10].time := 3600.0, [36].log_data[10].valid := 1, [36].log_data[11].time := 3600.0, [36].log_data[11].valid := 1, [36].log_data[12].min := 1.0, [36].log_data[12].max := 1.0, [36].log_data[12].total := 3600.0, [36].log_data[12].time := 3600.0, [36].log_data[12].valid := 1, [36].log_data[13].min := 1.0, [36].log_data[13].max := 1.0, [36].log_data[13].total := 3600.0, [36].log_data[13].time := 3600.0, [36].log_data[13].valid := 1, [36].log_data[14].time := 3600.0, [36].log_data[14].valid := 1, [36].log_data[15].time := 3600.0, [36].log_data[15].valid := 1, [36].log_data[16].time := 3600.0, [36].log_data[16].valid := 1, [36].log_data[17].min := 1.0, [36].log_data[17].max := 1.0, [36].log_data[17].total := 3600.0, [36].log_data[17].time := 3600.0, [36].log_data[17].valid := 1, [36].log_data[18].time := 3600.0, [36].log_data[18].valid := 1, [36].log_data[19].time := 3600.0, [36].log_data[19].valid := 1, [36].log_data[20].time := 3600.0, [36].log_data[20].valid := 1, [36].log_data[21].min := 1.0, [36].log_data[21].max := 1.0, [36].log_data[21].total := 3600.0, [36].log_data[21].time := 3600.0, [36].log_data[21].valid := 1, [36].log_data[22].time := 3600.0,
        [36].log_data[22].valid := 1, [36].log_data[23].time := 3600.0, [36].log_data[23].valid := 1, [36].log_data[24].time := 3600.0, [36].log_data[24].valid := 1, [36].log_data[25].time := 3600.0, [36].log_data[25].valid := 1, [36].log_data[26].time := 3600.0, [36].log_data[26].valid := 1, [36].log_data[27].time := 3600.0, [36].log_data[27].valid := 1, [36].log_data[28].time := 3600.0, [36].log_data[28].valid := 1, [36].log_data[29].min := 1.0, [36].log_data[29].max := 1.0, [36].log_data[29].total := 3600.0, [36].log_data[29].time := 3600.0, [36].log_data[29].valid := 1, [36].log_data[30].min := 1.0, [36].log_data[30].max := 1.0, [36].log_data[30].total := 3600.0, [36].log_data[30].time := 3600.0, [36].log_data[30].valid := 1, [36].log_data[31].max := 1.0, [36].log_data[31].total := 1629.998, [36].log_data[31].time := 3600.0, [36].log_data[31].maxminute := 2, [36].log_data[31].valid := 1, [36].log_data[32].max := 1.0, [36].log_data[32].total := 1440.749, [36].log_data[32].time := 3600.0, [36].log_data[32].minminute := 1, [36].log_data[32].valid := 1, [36].log_data[33].time := 3600.0, [36].log_data[33].valid := 1, [36].log_data[34].time := 3600.0, [36].log_data[34].valid := 1, [36].log_data[35].max := 1.0, [36].log_data[35].total := 1475.498, [36].log_data[35].time := 3600.0, [36].log_data[35].minminute := 6, [36].log_data[35].valid := 1, [36].log_data[36].max := 1.0, [36].log_data[36].total := 1629.7471, [36].log_data[36].time := 3600.0, [36].log_data[36].maxminute := 7, [36].log_data[36].valid := 1, [36].log_data[37].time := 3600.0, [36].log_data[37].valid := 1, [36].log_data[38].time := 3600.0, [36].log_data[38].valid := 1, [36].log_data[39].min := 0.9947063, [36].log_data[39].max := 1.0062482, [36].log_data[39].total := 3605.5598, [36].log_data[39].time := 3600.0, [36].log_data[39].minminute := 12, [36].log_data[39].maxminute := 47, [36].log_data[39].valid := 1, [36].log_data[40].min := 7.5700884, [36].log_data[40].max := 7.592072,
        [36].log_data[40].total := 27300.482, [36].log_data[40].time := 3600.0, [36].log_data[40].minminute := 28, [36].log_data[40].maxminute := 36, [36].log_data[40].valid := 1, [36].log_data[41].min := 0.037261963, [36].log_data[41].max := 0.048843265, [36].log_data[41].total := 159.3191, [36].log_data[41].time := 3600.0, [36].log_data[41].maxminute := 28, [36].log_data[41].valid := 1, [36].log_data[42].min := 2.292467, [36].log_data[42].max := 2.297178, [36].log_data[42].total := 8262.197, [36].log_data[42].time := 3600.0, [36].log_data[42].minminute := 30, [36].log_data[42].maxminute := 6, [36].log_data[42].valid := 1, [36].log_data[43].min := -0.27999878, [36].log_data[43].max := -0.26000214, [36].log_data[43].total := -949.0952, [36].log_data[43].time := 3600.0, [36].log_data[43].valid := 1, [36].log_data[44].min := -0.30000305, [36].log_data[44].max := -0.30000305, [36].log_data[44].total := -1080.0911, [36].log_data[44].time := 3600.0, [36].log_data[44].valid := 1, [36].log_data[45].time := 3600.0, [36].log_data[45].valid := 1, [36].log_data[46].time := 3600.0, [36].log_data[46].valid := 1, [36].log_data[47].time := 3600.0, [36].log_data[47].valid := 1, [36].log_data[48].min := 6.5821533, [36].log_data[48].max := 6.7852364, [36].log_data[48].total := 24176.883, [36].log_data[48].time := 3600.0, [36].log_data[48].minminute := 13, [36].log_data[48].maxminute := 29, [36].log_data[48].valid := 1, [36].log_data[49].min := 7.0024657, [36].log_data[49].max := 9.6019535, [36].log_data[49].total := 30474.594, [36].log_data[49].time := 3600.0, [36].log_data[49].minminute := 10, [36].log_data[49].maxminute := 59, [36].log_data[49].valid := 1, [36].log_data[50].min := 2.0887165, [36].log_data[50].max := 2.1765766, [36].log_data[50].total := 7677.809, [36].log_data[50].time := 3600.0, [36].log_data[50].minminute := 59, [36].log_data[50].valid := 1, [36].log_data[51].time := 3600.0, [36].log_data[51].valid := 1, [36].log_data[52].min := -3.1200027, [36].log_data[52].max := 0.11999512, [36].log_data[52].total := -7562.2544, [36].log_data[52].time := 3600.0,
        [36].log_data[52].minminute := 24, [36].log_data[52].maxminute := 1, [36].log_data[52].valid := 1, [36].log_data[53].min := -2.4800034, [36].log_data[53].max := 0.22000122, [36].log_data[53].total := -7105.2676, [36].log_data[53].time := 3600.0, [36].log_data[53].minminute := 5, [36].log_data[53].maxminute := 7, [36].log_data[53].valid := 1, [36].log_data[54].max := 0.557, [36].log_data[54].total := 1217.6827, [36].log_data[54].time := 3600.0, [36].log_data[54].minminute := 1, [36].log_data[54].maxminute := 24, [36].log_data[54].valid := 1, [36].log_data[55].max := 0.5285, [36].log_data[55].total := 1233.2991, [36].log_data[55].time := 3600.0, [36].log_data[55].minminute := 6, [36].log_data[55].maxminute := 18, [36].log_data[55].valid := 1, [36].log_data[56].min := 0.16008857, [36].log_data[56].max := 0.1605204, [36].log_data[56].total := 577.0054, [36].log_data[56].time := 3600.0, [36].log_data[56].minminute := 19, [36].log_data[56].valid := 1, [36].log_data[57].min := 0.29101494, [36].log_data[57].max := 0.29313487, [36].log_data[57].total := 1049.9497, [36].log_data[57].time := 3600.0, [36].log_data[57].minminute := 30, [36].log_data[57].maxminute := 1, [36].log_data[57].valid := 1, [36].log_data[58].time := 3600.0, [36].log_data[58].valid := 1, [36].log_data[59].time := 3600.0, [36].log_data[59].valid := 1, [36].log_data[60].valid := 1, [36].log_data[61].valid := 1, [36].log_data[62].valid := 1, [36].log_data[63].valid := 1, [36].log_data[64].valid := 1, [36].log_data[65].valid := 1, [36].log_data[66].valid := 1, [36].log_data[67].valid := 1, [36].log_data[68].valid := 1, [36].log_data[69].valid := 1, [36].log_data[70].valid := 1, [36].log_data[71].valid := 1, [36].log_data[72].valid := 1, [36].log_data[73].valid := 1, [36].log_data[74].valid := 1, [36].log_data[75].valid := 1, [36].log_data[76].valid := 1, [36].log_data[77].valid := 1, [36].log_data[78].valid := 1, [36].log_data[79].valid := 1, [36].log_data[80].valid := 1,
        [36].log_data[81].valid := 1, [36].log_data[82].valid := 1, [36].log_data[83].valid := 1, [36].log_data[84].valid := 1, [36].log_data[85].valid := 1, [36].log_data[86].valid := 1, [36].log_data[87].valid := 1, [36].log_data[88].valid := 1, [36].log_data[89].valid := 1, [36].log_data[90].valid := 1, [36].log_data[91].valid := 1, [36].log_data[92].valid := 1, [36].log_data[93].valid := 1, [36].log_data[94].valid := 1, [36].log_data[95].valid := 1, [36].log_data[96].valid := 1, [36].log_data[97].valid := 1, [36].log_data[98].valid := 1, [36].log_data[99].valid := 1, [36].log_data[100].valid := 1, [36].log_data[101].valid := 1, [36].log_data[102].valid := 1, [36].log_data[103].valid := 1, [36].log_data[104].valid := 1, [36].log_data[105].valid := 1, [36].log_data[106].valid := 1, [36].log_data[107].valid := 1, [36].log_data[108].valid := 1, [36].log_data[109].valid := 1, [36].log_data[110].valid := 1, [36].log_data[111].valid := 1, [36].log_data[112].valid := 1, [36].log_data[113].valid := 1, [36].log_data[114].valid := 1, [36].log_data[115].valid := 1, [36].log_data[116].valid := 1, [36].log_data[117].valid := 1, [36].log_data[118].valid := 1, [36].log_data[119].valid := 1, [36].log_data[120].valid := 1, [36].log_data[121].valid := 1, [36].log_data[122].valid := 1, [36].log_data[123].valid := 1, [36].log_data[124].valid := 1, [36].time.Year := 2023, [36].time.Month := 1, [36].time.Day := 14, [36].time.Hour := 15, [36].time.Minute := 59, [36].time.Second := 59, [37].log_data[0].min := 1.0, [37].log_data[0].max := 1.0, [37].log_data[0].total := 3600.0, [37].log_data[0].time := 3600.0, [37].log_data[0].valid := 1, [37].log_data[1].max := 1.0, [37].log_data[1].total := 547.0, [37].log_data[1].time := 3600.0, [37].log_data[1].maxminute := 30, [37].log_data[1].valid := 1,
        [37].log_data[2].max := 1.0, [37].log_data[2].total := 543.5, [37].log_data[2].time := 3600.0, [37].log_data[2].maxminute := 30, [37].log_data[2].valid := 1, [37].log_data[3].time := 3600.0, [37].log_data[3].valid := 1, [37].log_data[4].time := 3600.0, [37].log_data[4].valid := 1, [37].log_data[5].max := 1.0, [37].log_data[5].total := 228.5, [37].log_data[5].time := 3600.0, [37].log_data[5].maxminute := 33, [37].log_data[5].valid := 1, [37].log_data[6].time := 3600.0, [37].log_data[6].valid := 1, [37].log_data[7].time := 3600.0, [37].log_data[7].valid := 1, [37].log_data[8].min := 1.0, [37].log_data[8].max := 1.0, [37].log_data[8].total := 3600.0, [37].log_data[8].time := 3600.0, [37].log_data[8].valid := 1, [37].log_data[9].min := 1.0, [37].log_data[9].max := 1.0, [37].log_data[9].total := 3600.0, [37].log_data[9].time := 3600.0, [37].log_data[9].valid := 1, [37].log_data[10].min := 1.0, [37].log_data[10].max := 1.0, [37].log_data[10].total := 3600.0, [37].log_data[10].time := 3600.0, [37].log_data[10].valid := 1, [37].log_data[11].time := 3600.0, [37].log_data[11].valid := 1, [37].log_data[12].min := 1.0, [37].log_data[12].max := 1.0, [37].log_data[12].total := 3600.0, [37].log_data[12].time := 3600.0, [37].log_data[12].valid := 1, [37].log_data[13].min := 1.0, [37].log_data[13].max := 1.0, [37].log_data[13].total := 3600.0, [37].log_data[13].time := 3600.0, [37].log_data[13].valid := 1, [37].log_data[14].time := 3600.0, [37].log_data[14].valid := 1, [37].log_data[15].time := 3600.0, [37].log_data[15].valid := 1, [37].log_data[16].time := 3600.0, [37].log_data[16].valid := 1, [37].log_data[17].min := 1.0, [37].log_data[17].max := 1.0, [37].log_data[17].total := 3600.0, [37].log_data[17].time := 3600.0, [37].log_data[17].valid := 1, [37].log_data[18].time := 3600.0, [37].log_data[18].valid := 1, [37].log_data[19].time := 3600.0, [37].log_data[19].valid := 1,
        [37].log_data[20].time := 3600.0, [37].log_data[20].valid := 1, [37].log_data[21].min := 1.0, [37].log_data[21].max := 1.0, [37].log_data[21].total := 3600.0, [37].log_data[21].time := 3600.0, [37].log_data[21].valid := 1, [37].log_data[22].time := 3600.0, [37].log_data[22].valid := 1, [37].log_data[23].time := 3600.0, [37].log_data[23].valid := 1, [37].log_data[24].time := 3600.0, [37].log_data[24].valid := 1, [37].log_data[25].time := 3600.0, [37].log_data[25].valid := 1, [37].log_data[26].time := 3600.0, [37].log_data[26].valid := 1, [37].log_data[27].time := 3600.0, [37].log_data[27].valid := 1, [37].log_data[28].time := 3600.0, [37].log_data[28].valid := 1, [37].log_data[29].min := 1.0, [37].log_data[29].max := 1.0, [37].log_data[29].total := 3600.0, [37].log_data[29].time := 3600.0, [37].log_data[29].valid := 1, [37].log_data[30].min := 1.0, [37].log_data[30].max := 1.0, [37].log_data[30].total := 3600.0, [37].log_data[30].time := 3600.0, [37].log_data[30].valid := 1, [37].log_data[31].max := 1.0, [37].log_data[31].total := 1629.998, [37].log_data[31].time := 3600.0, [37].log_data[31].maxminute := 6, [37].log_data[31].valid := 1, [37].log_data[32].max := 1.0, [37].log_data[32].total := 1440.998, [37].log_data[32].time := 3600.0, [37].log_data[32].minminute := 4, [37].log_data[32].valid := 1, [37].log_data[33].time := 3600.0, [37].log_data[33].valid := 1, [37].log_data[34].time := 3600.0, [37].log_data[34].valid := 1, [37].log_data[35].max := 1.0, [37].log_data[35].total := 1629.7471, [37].log_data[35].time := 3600.0, [37].log_data[35].valid := 1, [37].log_data[36].max := 1.0, [37].log_data[36].total := 1494.2471, [37].log_data[36].time := 3600.0, [37].log_data[36].maxminute := 11, [37].log_data[36].valid := 1, [37].log_data[37].max := 7.3518314, [37].log_data[37].total := 3482.6306, [37].log_data[37].time := 3600.0, [37].log_data[37].maxminute := 33, [37].log_data[37].valid := 1, [37].log_data[38].time := 3600.0,
        [37].log_data[38].valid := 1, [37].log_data[39].min := 0.9945885, [37].log_data[39].max := 1.0230899, [37].log_data[39].total := 3612.0276, [37].log_data[39].time := 3600.0, [37].log_data[39].minminute := 19, [37].log_data[39].maxminute := 37, [37].log_data[39].valid := 1, [37].log_data[40].min := 7.5788817, [37].log_data[40].max := 7.585202, [37].log_data[40].total := 27304.906, [37].log_data[40].time := 3600.0, [37].log_data[40].minminute := 51, [37].log_data[40].maxminute := 1, [37].log_data[40].valid := 1, [37].log_data[41].min := 0.028232668, [37].log_data[41].max := 0.052769043, [37].log_data[41].total := 147.9353, [37].log_data[41].time := 3600.0, [37].log_data[41].minminute := 33, [37].log_data[41].maxminute := 5, [37].log_data[41].valid := 1, [37].log_data[42].min := 2.292467, [37].log_data[42].max := 2.297178, [37].log_data[42].total := 8262.205, [37].log_data[42].time := 3600.0, [37].log_data[42].minminute := 14, [37].log_data[42].maxminute := 34, [37].log_data[42].valid := 1, [37].log_data[43].min := -0.27999878, [37].log_data[43].max := -0.26000214, [37].log_data[43].total := -994.96844, [37].log_data[43].time := 3600.0, [37].log_data[43].valid := 1, [37].log_data[44].min := -0.3199997, [37].log_data[44].max := -0.30000305, [37].log_data[44].total := -1092.3223, [37].log_data[44].time := 3600.0, [37].log_data[44].minminute := 4, [37].log_data[44].valid := 1, [37].log_data[45].time := 3600.0, [37].log_data[45].valid := 1, [37].log_data[46].time := 3600.0, [37].log_data[46].valid := 1, [37].log_data[47].time := 3600.0, [37].log_data[47].valid := 1, [37].log_data[48].min := 6.595069, [37].log_data[48].max := 6.924289, [37].log_data[48].total := 24282.354, [37].log_data[48].time := 3600.0, [37].log_data[48].minminute := 59, [37].log_data[48].maxminute := 39, [37].log_data[48].valid := 1, [37].log_data[49].min := 7.082945, [37].log_data[49].max := 9.652988, [37].log_data[49].total := 31927.703, [37].log_data[49].time := 3600.0, [37].log_data[49].minminute := 59, [37].log_data[49].maxminute := 33, [37].log_data[49].valid := 1,
        [37].log_data[50].min := 2.0451398, [37].log_data[50].max := 2.1463084, [37].log_data[50].total := 7538.133, [37].log_data[50].time := 3600.0, [37].log_data[50].minminute := 30, [37].log_data[50].maxminute := 39, [37].log_data[50].valid := 1, [37].log_data[51].time := 3600.0, [37].log_data[51].valid := 1, [37].log_data[52].min := -3.0200043, [37].log_data[52].max := 0.11999512, [37].log_data[52].total := -7619.2183, [37].log_data[52].time := 3600.0, [37].log_data[52].minminute := 6, [37].log_data[52].maxminute := 4, [37].log_data[52].valid := 1, [37].log_data[53].min := -2.6600037, [37].log_data[53].max := 0.2400055, [37].log_data[53].total := -7223.1343, [37].log_data[53].time := 3600.0, [37].log_data[53].minminute := 21, [37].log_data[53].maxminute := 31, [37].log_data[53].valid := 1, [37].log_data[54].max := 0.555, [37].log_data[54].total := 1217.5787, [37].log_data[54].time := 3600.0, [37].log_data[54].minminute := 4, [37].log_data[54].maxminute := 6, [37].log_data[54].valid := 1, [37].log_data[55].max := 0.52250004, [37].log_data[55].total := 1238.3247, [37].log_data[55].time := 3600.0, [37].log_data[55].maxminute := 21, [37].log_data[55].valid := 1, [37].log_data[56].min := 0.16012783, [37].log_data[56].max := 0.1605204, [37].log_data[56].total := 576.9781, [37].log_data[56].time := 3600.0, [37].log_data[56].minminute := 5, [37].log_data[56].valid := 1, [37].log_data[57].min := 0.29101494, [37].log_data[57].max := 0.29144678, [37].log_data[57].total := 1048.2297, [37].log_data[57].time := 3600.0, [37].log_data[57].minminute := 5, [37].log_data[57].maxminute := 12, [37].log_data[57].valid := 1, [37].log_data[58].time := 3600.0, [37].log_data[58].valid := 1, [37].log_data[59].time := 3600.0, [37].log_data[59].valid := 1, [37].log_data[60].valid := 1, [37].log_data[61].valid := 1, [37].log_data[62].valid := 1, [37].log_data[63].valid := 1, [37].log_data[64].valid := 1, [37].log_data[65].valid := 1, [37].log_data[66].valid := 1, [37].log_data[67].valid := 1, [37].log_data[68].valid := 1,
        [37].log_data[69].valid := 1, [37].log_data[70].valid := 1, [37].log_data[71].valid := 1, [37].log_data[72].valid := 1, [37].log_data[73].valid := 1, [37].log_data[74].valid := 1, [37].log_data[75].valid := 1, [37].log_data[76].valid := 1, [37].log_data[77].valid := 1, [37].log_data[78].valid := 1, [37].log_data[79].valid := 1, [37].log_data[80].valid := 1, [37].log_data[81].valid := 1, [37].log_data[82].valid := 1, [37].log_data[83].valid := 1, [37].log_data[84].valid := 1, [37].log_data[85].valid := 1, [37].log_data[86].valid := 1, [37].log_data[87].valid := 1, [37].log_data[88].valid := 1, [37].log_data[89].valid := 1, [37].log_data[90].valid := 1, [37].log_data[91].valid := 1, [37].log_data[92].valid := 1, [37].log_data[93].valid := 1, [37].log_data[94].valid := 1, [37].log_data[95].valid := 1, [37].log_data[96].valid := 1, [37].log_data[97].valid := 1, [37].log_data[98].valid := 1, [37].log_data[99].valid := 1, [37].log_data[100].valid := 1, [37].log_data[101].valid := 1, [37].log_data[102].valid := 1, [37].log_data[103].valid := 1, [37].log_data[104].valid := 1, [37].log_data[105].valid := 1, [37].log_data[106].valid := 1, [37].log_data[107].valid := 1, [37].log_data[108].valid := 1, [37].log_data[109].valid := 1, [37].log_data[110].valid := 1, [37].log_data[111].valid := 1, [37].log_data[112].valid := 1, [37].log_data[113].valid := 1, [37].log_data[114].valid := 1, [37].log_data[115].valid := 1, [37].log_data[116].valid := 1, [37].log_data[117].valid := 1, [37].log_data[118].valid := 1, [37].log_data[119].valid := 1, [37].log_data[120].valid := 1, [37].log_data[121].valid := 1, [37].log_data[122].valid := 1, [37].log_data[123].valid := 1, [37].log_data[124].valid := 1, [37].time.Year := 2023, [37].time.Month := 1, [37].time.Day := 14, [37].time.Hour := 16,
        [37].time.Minute := 59, [37].time.Second := 59, [38].log_data[0].min := 1.0, [38].log_data[0].max := 1.0, [38].log_data[0].total := 3600.0, [38].log_data[0].time := 3600.0, [38].log_data[0].valid := 1, [38].log_data[1].time := 3600.0, [38].log_data[1].valid := 1, [38].log_data[2].time := 3600.0, [38].log_data[2].valid := 1, [38].log_data[3].time := 3600.0, [38].log_data[3].valid := 1, [38].log_data[4].time := 3600.0, [38].log_data[4].valid := 1, [38].log_data[5].time := 3600.0, [38].log_data[5].valid := 1, [38].log_data[6].time := 3600.0, [38].log_data[6].valid := 1, [38].log_data[7].time := 3600.0, [38].log_data[7].valid := 1, [38].log_data[8].min := 1.0, [38].log_data[8].max := 1.0, [38].log_data[8].total := 3600.0, [38].log_data[8].time := 3600.0, [38].log_data[8].valid := 1, [38].log_data[9].min := 1.0, [38].log_data[9].max := 1.0, [38].log_data[9].total := 3600.0, [38].log_data[9].time := 3600.0, [38].log_data[9].valid := 1, [38].log_data[10].min := 1.0, [38].log_data[10].max := 1.0, [38].log_data[10].total := 3600.0, [38].log_data[10].time := 3600.0, [38].log_data[10].valid := 1, [38].log_data[11].time := 3600.0, [38].log_data[11].valid := 1, [38].log_data[12].min := 1.0, [38].log_data[12].max := 1.0, [38].log_data[12].total := 3600.0, [38].log_data[12].time := 3600.0, [38].log_data[12].valid := 1, [38].log_data[13].min := 1.0, [38].log_data[13].max := 1.0, [38].log_data[13].total := 3600.0, [38].log_data[13].time := 3600.0, [38].log_data[13].valid := 1, [38].log_data[14].time := 3600.0, [38].log_data[14].valid := 1, [38].log_data[15].time := 3600.0, [38].log_data[15].valid := 1, [38].log_data[16].time := 3600.0, [38].log_data[16].valid := 1, [38].log_data[17].min := 1.0, [38].log_data[17].max := 1.0, [38].log_data[17].total := 3600.0, [38].log_data[17].time := 3600.0, [38].log_data[17].valid := 1, [38].log_data[18].time := 3600.0,
        [38].log_data[18].valid := 1, [38].log_data[19].time := 3600.0, [38].log_data[19].valid := 1, [38].log_data[20].time := 3600.0, [38].log_data[20].valid := 1, [38].log_data[21].min := 1.0, [38].log_data[21].max := 1.0, [38].log_data[21].total := 3600.0, [38].log_data[21].time := 3600.0, [38].log_data[21].valid := 1, [38].log_data[22].time := 3600.0, [38].log_data[22].valid := 1, [38].log_data[23].time := 3600.0, [38].log_data[23].valid := 1, [38].log_data[24].time := 3600.0, [38].log_data[24].valid := 1, [38].log_data[25].time := 3600.0, [38].log_data[25].valid := 1, [38].log_data[26].time := 3600.0, [38].log_data[26].valid := 1, [38].log_data[27].time := 3600.0, [38].log_data[27].valid := 1, [38].log_data[28].time := 3600.0, [38].log_data[28].valid := 1, [38].log_data[29].min := 1.0, [38].log_data[29].max := 1.0, [38].log_data[29].total := 3600.0, [38].log_data[29].time := 3600.0, [38].log_data[29].valid := 1, [38].log_data[30].min := 1.0, [38].log_data[30].max := 1.0, [38].log_data[30].total := 3600.0, [38].log_data[30].time := 3600.0, [38].log_data[30].valid := 1, [38].log_data[31].max := 1.0, [38].log_data[31].total := 1602.7471, [38].log_data[31].time := 3600.0, [38].log_data[31].maxminute := 9, [38].log_data[31].valid := 1, [38].log_data[32].max := 1.0, [38].log_data[32].total := 1556.249, [38].log_data[32].time := 3600.0, [38].log_data[32].minminute := 7, [38].log_data[32].valid := 1, [38].log_data[33].time := 3600.0, [38].log_data[33].valid := 1, [38].log_data[34].time := 3600.0, [38].log_data[34].valid := 1, [38].log_data[35].max := 1.0, [38].log_data[35].total := 1629.998, [38].log_data[35].time := 3600.0, [38].log_data[35].maxminute := 3, [38].log_data[35].valid := 1, [38].log_data[36].max := 1.0, [38].log_data[36].total := 1440.498, [38].log_data[36].time := 3600.0, [38].log_data[36].minminute := 2, [38].log_data[36].valid := 1, [38].log_data[37].time := 3600.0, [38].log_data[37].valid := 1,
        [38].log_data[38].time := 3600.0, [38].log_data[38].valid := 1, [38].log_data[39].min := 0.9965906, [38].log_data[39].max := 1.0082504, [38].log_data[39].total := 3611.5464, [38].log_data[39].time := 3600.0, [38].log_data[39].minminute := 50, [38].log_data[39].maxminute := 53, [38].log_data[39].valid := 1, [38].log_data[40].min := 7.5731106, [38].log_data[40].max := 7.590698, [38].log_data[40].total := 27303.076, [38].log_data[40].time := 3600.0, [38].log_data[40].minminute := 55, [38].log_data[40].maxminute := 58, [38].log_data[40].valid := 1, [38].log_data[41].min := 0.026858643, [38].log_data[41].max := 0.04864697, [38].log_data[41].total := 132.5628, [38].log_data[41].time := 3600.0, [38].log_data[41].minminute := 25, [38].log_data[41].maxminute := 8, [38].log_data[41].valid := 1, [38].log_data[42].min := 2.292585, [38].log_data[42].max := 2.2970603, [38].log_data[42].total := 8262.251, [38].log_data[42].time := 3600.0, [38].log_data[42].minminute := 26, [38].log_data[42].maxminute := 20, [38].log_data[42].valid := 1, [38].log_data[43].min := -0.27999878, [38].log_data[43].max := -0.26000214, [38].log_data[43].total := -1007.8563, [38].log_data[43].time := 3600.0, [38].log_data[43].maxminute := 1, [38].log_data[43].valid := 1, [38].log_data[44].min := -0.3199997, [38].log_data[44].max := -0.30000305, [38].log_data[44].total := -1131.83, [38].log_data[44].time := 3600.0, [38].log_data[44].valid := 1, [38].log_data[45].time := 3600.0, [38].log_data[45].valid := 1, [38].log_data[46].time := 3600.0, [38].log_data[46].valid := 1, [38].log_data[47].time := 3600.0, [38].log_data[47].valid := 1, [38].log_data[48].min := 6.585176, [38].log_data[48].max := 6.784961, [38].log_data[48].total := 24251.959, [38].log_data[48].time := 3600.0, [38].log_data[48].minminute := 1, [38].log_data[48].maxminute := 16, [38].log_data[48].valid := 1, [38].log_data[49].min := 7.100415, [38].log_data[49].max := 9.636696, [38].log_data[49].total := 32306.947, [38].log_data[49].time := 3600.0, [38].log_data[49].maxminute := 53, [38].log_data[49].valid := 1,
        [38].log_data[50].min := 2.038309, [38].log_data[50].max := 2.1245203, [38].log_data[50].total := 7495.8105, [38].log_data[50].time := 3600.0, [38].log_data[50].minminute := 59, [38].log_data[50].valid := 1, [38].log_data[51].time := 3600.0, [38].log_data[51].valid := 1, [38].log_data[52].min := -3.0, [38].log_data[52].max := 0.11999512, [38].log_data[52].total := -7944.188, [38].log_data[52].time := 3600.0, [38].log_data[52].minminute := 30, [38].log_data[52].maxminute := 18, [38].log_data[52].valid := 1, [38].log_data[53].min := -2.5, [38].log_data[53].max := 0.2599945, [38].log_data[53].total := -7136.765, [38].log_data[53].time := 3600.0, [38].log_data[53].minminute := 21, [38].log_data[53].maxminute := 24, [38].log_data[53].valid := 1, [38].log_data[54].max := 0.5715, [38].log_data[54].total := 1254.9435, [38].log_data[54].time := 3600.0, [38].log_data[54].minminute := 7, [38].log_data[54].maxminute := 30, [38].log_data[54].valid := 1, [38].log_data[55].max := 0.538, [38].log_data[55].total := 1217.4385, [38].log_data[55].time := 3600.0, [38].log_data[55].minminute := 2, [38].log_data[55].maxminute := 35, [38].log_data[55].valid := 1, [38].log_data[56].min := 0.16008857, [38].log_data[56].max := 0.16055967, [38].log_data[56].total := 577.07654, [38].log_data[56].time := 3600.0, [38].log_data[56].minminute := 9, [38].log_data[56].maxminute := 27, [38].log_data[56].valid := 1, [38].log_data[57].min := 0.28928754, [38].log_data[57].max := 0.29121122, [38].log_data[57].total := 1042.6053, [38].log_data[57].time := 3600.0, [38].log_data[57].minminute := 10, [38].log_data[57].valid := 1, [38].log_data[58].time := 3600.0, [38].log_data[58].valid := 1, [38].log_data[59].time := 3600.0, [38].log_data[59].valid := 1, [38].log_data[60].valid := 1, [38].log_data[61].valid := 1, [38].log_data[62].valid := 1, [38].log_data[63].valid := 1, [38].log_data[64].valid := 1, [38].log_data[65].valid := 1, [38].log_data[66].valid := 1, [38].log_data[67].valid := 1, [38].log_data[68].valid := 1,
        [38].log_data[69].valid := 1, [38].log_data[70].valid := 1, [38].log_data[71].valid := 1, [38].log_data[72].valid := 1, [38].log_data[73].valid := 1, [38].log_data[74].valid := 1, [38].log_data[75].valid := 1, [38].log_data[76].valid := 1, [38].log_data[77].valid := 1, [38].log_data[78].valid := 1, [38].log_data[79].valid := 1, [38].log_data[80].valid := 1, [38].log_data[81].valid := 1, [38].log_data[82].valid := 1, [38].log_data[83].valid := 1, [38].log_data[84].valid := 1, [38].log_data[85].valid := 1, [38].log_data[86].valid := 1, [38].log_data[87].valid := 1, [38].log_data[88].valid := 1, [38].log_data[89].valid := 1, [38].log_data[90].valid := 1, [38].log_data[91].valid := 1, [38].log_data[92].valid := 1, [38].log_data[93].valid := 1, [38].log_data[94].valid := 1, [38].log_data[95].valid := 1, [38].log_data[96].valid := 1, [38].log_data[97].valid := 1, [38].log_data[98].valid := 1, [38].log_data[99].valid := 1, [38].log_data[100].valid := 1, [38].log_data[101].valid := 1, [38].log_data[102].valid := 1, [38].log_data[103].valid := 1, [38].log_data[104].valid := 1, [38].log_data[105].valid := 1, [38].log_data[106].valid := 1, [38].log_data[107].valid := 1, [38].log_data[108].valid := 1, [38].log_data[109].valid := 1, [38].log_data[110].valid := 1, [38].log_data[111].valid := 1, [38].log_data[112].valid := 1, [38].log_data[113].valid := 1, [38].log_data[114].valid := 1, [38].log_data[115].valid := 1, [38].log_data[116].valid := 1, [38].log_data[117].valid := 1, [38].log_data[118].valid := 1, [38].log_data[119].valid := 1, [38].log_data[120].valid := 1, [38].log_data[121].valid := 1, [38].log_data[122].valid := 1, [38].log_data[123].valid := 1, [38].log_data[124].valid := 1, [38].time.Year := 2023, [38].time.Month := 1, [38].time.Day := 14, [38].time.Hour := 17,
        [38].time.Minute := 59, [38].time.Second := 59, [39].log_data[0].min := 1.0, [39].log_data[0].max := 1.0, [39].log_data[0].total := 3600.0, [39].log_data[0].time := 3600.0, [39].log_data[0].valid := 1, [39].log_data[1].max := 1.0, [39].log_data[1].total := 541.5, [39].log_data[1].time := 3600.0, [39].log_data[1].maxminute := 11, [39].log_data[1].valid := 1, [39].log_data[2].max := 1.0, [39].log_data[2].total := 538.0, [39].log_data[2].time := 3600.0, [39].log_data[2].maxminute := 11, [39].log_data[2].valid := 1, [39].log_data[3].time := 3600.0, [39].log_data[3].valid := 1, [39].log_data[4].time := 3600.0, [39].log_data[4].valid := 1, [39].log_data[5].max := 1.0, [39].log_data[5].total := 235.5, [39].log_data[5].time := 3600.0, [39].log_data[5].maxminute := 13, [39].log_data[5].valid := 1, [39].log_data[6].time := 3600.0, [39].log_data[6].valid := 1, [39].log_data[7].time := 3600.0, [39].log_data[7].valid := 1, [39].log_data[8].min := 1.0, [39].log_data[8].max := 1.0, [39].log_data[8].total := 3600.0, [39].log_data[8].time := 3600.0, [39].log_data[8].valid := 1, [39].log_data[9].min := 1.0, [39].log_data[9].max := 1.0, [39].log_data[9].total := 3600.0, [39].log_data[9].time := 3600.0, [39].log_data[9].valid := 1, [39].log_data[10].min := 1.0, [39].log_data[10].max := 1.0, [39].log_data[10].total := 3600.0, [39].log_data[10].time := 3600.0, [39].log_data[10].valid := 1, [39].log_data[11].time := 3600.0, [39].log_data[11].valid := 1, [39].log_data[12].min := 1.0, [39].log_data[12].max := 1.0, [39].log_data[12].total := 3600.0, [39].log_data[12].time := 3600.0, [39].log_data[12].valid := 1, [39].log_data[13].min := 1.0, [39].log_data[13].max := 1.0, [39].log_data[13].total := 3600.0, [39].log_data[13].time := 3600.0, [39].log_data[13].valid := 1, [39].log_data[14].time := 3600.0, [39].log_data[14].valid := 1, [39].log_data[15].time := 3600.0,
        [39].log_data[15].valid := 1, [39].log_data[16].time := 3600.0, [39].log_data[16].valid := 1, [39].log_data[17].min := 1.0, [39].log_data[17].max := 1.0, [39].log_data[17].total := 3600.0, [39].log_data[17].time := 3600.0, [39].log_data[17].valid := 1, [39].log_data[18].time := 3600.0, [39].log_data[18].valid := 1, [39].log_data[19].time := 3600.0, [39].log_data[19].valid := 1, [39].log_data[20].time := 3600.0, [39].log_data[20].valid := 1, [39].log_data[21].min := 1.0, [39].log_data[21].max := 1.0, [39].log_data[21].total := 3600.0, [39].log_data[21].time := 3600.0, [39].log_data[21].valid := 1, [39].log_data[22].time := 3600.0, [39].log_data[22].valid := 1, [39].log_data[23].time := 3600.0, [39].log_data[23].valid := 1, [39].log_data[24].time := 3600.0, [39].log_data[24].valid := 1, [39].log_data[25].time := 3600.0, [39].log_data[25].valid := 1, [39].log_data[26].time := 3600.0, [39].log_data[26].valid := 1, [39].log_data[27].time := 3600.0, [39].log_data[27].valid := 1, [39].log_data[28].time := 3600.0, [39].log_data[28].valid := 1, [39].log_data[29].min := 1.0, [39].log_data[29].max := 1.0, [39].log_data[29].total := 3600.0, [39].log_data[29].time := 3600.0, [39].log_data[29].valid := 1, [39].log_data[30].min := 1.0, [39].log_data[30].max := 1.0, [39].log_data[30].total := 3600.0, [39].log_data[30].time := 3600.0, [39].log_data[30].valid := 1, [39].log_data[31].max := 1.0, [39].log_data[31].total := 1440.998, [39].log_data[31].time := 3600.0, [39].log_data[31].valid := 1, [39].log_data[32].max := 1.0, [39].log_data[32].total := 1629.998, [39].log_data[32].time := 3600.0, [39].log_data[32].maxminute := 1, [39].log_data[32].valid := 1, [39].log_data[33].time := 3600.0, [39].log_data[33].valid := 1, [39].log_data[34].time := 3600.0, [39].log_data[34].valid := 1, [39].log_data[35].max := 1.0, [39].log_data[35].total := 1629.749, [39].log_data[35].time := 3600.0, [39].log_data[35].maxminute := 6,
        [39].log_data[35].valid := 1, [39].log_data[36].max := 1.0, [39].log_data[36].total := 1440.7471, [39].log_data[36].time := 3600.0, [39].log_data[36].minminute := 5, [39].log_data[36].valid := 1, [39].log_data[37].max := 7.5807066, [39].log_data[37].total := 3563.3938, [39].log_data[37].time := 3600.0, [39].log_data[37].maxminute := 13, [39].log_data[37].valid := 1, [39].log_data[38].time := 3600.0, [39].log_data[38].valid := 1, [39].log_data[39].min := 0.9961195, [39].log_data[39].max := 1.0210879, [39].log_data[39].total := 3615.3127, [39].log_data[39].time := 3600.0, [39].log_data[39].minminute := 8, [39].log_data[39].maxminute := 17, [39].log_data[39].valid := 1, [39].log_data[40].min := 7.5758586, [39].log_data[40].max := 7.590698, [39].log_data[40].total := 27304.164, [39].log_data[40].time := 3600.0, [39].log_data[40].minminute := 30, [39].log_data[40].maxminute := 8, [39].log_data[40].valid := 1, [39].log_data[41].min := 0.03412134, [39].log_data[41].max := 0.057872556, [39].log_data[41].total := 167.72084, [39].log_data[41].time := 3600.0, [39].log_data[41].minminute := 3, [39].log_data[41].maxminute := 19, [39].log_data[41].valid := 1, [39].log_data[42].min := 2.292585, [39].log_data[42].max := 2.2970603, [39].log_data[42].total := 8262.185, [39].log_data[42].time := 3600.0, [39].log_data[42].minminute := 22, [39].log_data[42].maxminute := 49, [39].log_data[42].valid := 1, [39].log_data[43].min := -0.27999878, [39].log_data[43].max := -0.27999878, [39].log_data[43].total := -1007.8613, [39].log_data[43].time := 3600.0, [39].log_data[43].valid := 1, [39].log_data[44].min := -0.3199997, [39].log_data[44].max := -0.30000305, [39].log_data[44].total := -1130.2772, [39].log_data[44].time := 3600.0, [39].log_data[44].valid := 1, [39].log_data[45].time := 3600.0, [39].log_data[45].valid := 1, [39].log_data[46].time := 3600.0, [39].log_data[46].valid := 1, [39].log_data[47].time := 3600.0, [39].log_data[47].valid := 1, [39].log_data[48].min := 6.576932, [39].log_data[48].max := 6.9388537, [39].log_data[48].total := 24207.21,
        [39].log_data[48].time := 3600.0, [39].log_data[48].minminute := 42, [39].log_data[48].maxminute := 19, [39].log_data[48].valid := 1, [39].log_data[49].min := 7.010906, [39].log_data[49].max := 9.6276655, [39].log_data[49].total := 29849.309, [39].log_data[49].time := 3600.0, [39].log_data[49].minminute := 36, [39].log_data[49].maxminute := 3, [39].log_data[49].valid := 1, [39].log_data[50].min := 2.0206428, [39].log_data[50].max := 2.1255803, [39].log_data[50].total := 7498.8916, [39].log_data[50].time := 3600.0, [39].log_data[50].minminute := 13, [39].log_data[50].maxminute := 20, [39].log_data[50].valid := 1, [39].log_data[51].time := 3600.0, [39].log_data[51].valid := 1, [39].log_data[52].min := -2.880005, [39].log_data[52].max := 0.11999512, [39].log_data[52].total := -7729.3506, [39].log_data[52].time := 3600.0, [39].log_data[52].minminute := 33, [39].log_data[52].valid := 1, [39].log_data[53].min := -2.5, [39].log_data[53].max := 0.19999695, [39].log_data[53].total := -7153.875, [39].log_data[53].time := 3600.0, [39].log_data[53].minminute := 18, [39].log_data[53].maxminute := 59, [39].log_data[53].valid := 1, [39].log_data[54].max := 0.52349997, [39].log_data[54].total := 1217.3593, [39].log_data[54].time := 3600.0, [39].log_data[54].maxminute := 54, [39].log_data[54].valid := 1, [39].log_data[55].max := 0.532, [39].log_data[55].total := 1217.3375, [39].log_data[55].time := 3600.0, [39].log_data[55].minminute := 5, [39].log_data[55].maxminute := 28, [39].log_data[55].valid := 1, [39].log_data[56].min := 0.16016708, [39].log_data[56].max := 0.16059892, [39].log_data[56].total := 577.1995, [39].log_data[56].time := 3600.0, [39].log_data[56].minminute := 8, [39].log_data[56].maxminute := 28, [39].log_data[56].valid := 1, [39].log_data[57].min := 0.28763872, [39].log_data[57].max := 0.28971943, [39].log_data[57].total := 1040.4707, [39].log_data[57].time := 3600.0, [39].log_data[57].minminute := 53, [39].log_data[57].maxminute := 1, [39].log_data[57].valid := 1, [39].log_data[58].time := 3600.0, [39].log_data[58].valid := 1,
        [39].log_data[59].time := 3600.0, [39].log_data[59].valid := 1, [39].log_data[60].valid := 1, [39].log_data[61].valid := 1, [39].log_data[62].valid := 1, [39].log_data[63].valid := 1, [39].log_data[64].valid := 1, [39].log_data[65].valid := 1, [39].log_data[66].valid := 1, [39].log_data[67].valid := 1, [39].log_data[68].valid := 1, [39].log_data[69].valid := 1, [39].log_data[70].valid := 1, [39].log_data[71].valid := 1, [39].log_data[72].valid := 1, [39].log_data[73].valid := 1, [39].log_data[74].valid := 1, [39].log_data[75].valid := 1, [39].log_data[76].valid := 1, [39].log_data[77].valid := 1, [39].log_data[78].valid := 1, [39].log_data[79].valid := 1, [39].log_data[80].valid := 1, [39].log_data[81].valid := 1, [39].log_data[82].valid := 1, [39].log_data[83].valid := 1, [39].log_data[84].valid := 1, [39].log_data[85].valid := 1, [39].log_data[86].valid := 1, [39].log_data[87].valid := 1, [39].log_data[88].valid := 1, [39].log_data[89].valid := 1, [39].log_data[90].valid := 1, [39].log_data[91].valid := 1, [39].log_data[92].valid := 1, [39].log_data[93].valid := 1, [39].log_data[94].valid := 1, [39].log_data[95].valid := 1, [39].log_data[96].valid := 1, [39].log_data[97].valid := 1, [39].log_data[98].valid := 1, [39].log_data[99].valid := 1, [39].log_data[100].valid := 1, [39].log_data[101].valid := 1, [39].log_data[102].valid := 1, [39].log_data[103].valid := 1, [39].log_data[104].valid := 1, [39].log_data[105].valid := 1, [39].log_data[106].valid := 1, [39].log_data[107].valid := 1, [39].log_data[108].valid := 1, [39].log_data[109].valid := 1, [39].log_data[110].valid := 1, [39].log_data[111].valid := 1, [39].log_data[112].valid := 1, [39].log_data[113].valid := 1, [39].log_data[114].valid := 1, [39].log_data[115].valid := 1, [39].log_data[116].valid := 1, [39].log_data[117].valid := 1,
        [39].log_data[118].valid := 1, [39].log_data[119].valid := 1, [39].log_data[120].valid := 1, [39].log_data[121].valid := 1, [39].log_data[122].valid := 1, [39].log_data[123].valid := 1, [39].log_data[124].valid := 1, [39].time.Year := 2023, [39].time.Month := 1, [39].time.Day := 14, [39].time.Hour := 18, [39].time.Minute := 59, [39].time.Second := 59, [40].log_data[0].min := 1.0, [40].log_data[0].max := 1.0, [40].log_data[0].total := 3600.0, [40].log_data[0].time := 3600.0, [40].log_data[0].valid := 1, [40].log_data[1].max := 1.0, [40].log_data[1].total := 566.0, [40].log_data[1].time := 3600.0, [40].log_data[1].maxminute := 36, [40].log_data[1].valid := 1, [40].log_data[2].max := 1.0, [40].log_data[2].total := 562.5, [40].log_data[2].time := 3600.0, [40].log_data[2].maxminute := 36, [40].log_data[2].valid := 1, [40].log_data[3].time := 3600.0, [40].log_data[3].valid := 1, [40].log_data[4].time := 3600.0, [40].log_data[4].valid := 1, [40].log_data[5].max := 1.0, [40].log_data[5].total := 222.0, [40].log_data[5].time := 3600.0, [40].log_data[5].maxminute := 38, [40].log_data[5].valid := 1, [40].log_data[6].time := 3600.0, [40].log_data[6].valid := 1, [40].log_data[7].time := 3600.0, [40].log_data[7].valid := 1, [40].log_data[8].min := 1.0, [40].log_data[8].max := 1.0, [40].log_data[8].total := 3600.0, [40].log_data[8].time := 3600.0, [40].log_data[8].valid := 1, [40].log_data[9].min := 1.0, [40].log_data[9].max := 1.0, [40].log_data[9].total := 3600.0, [40].log_data[9].time := 3600.0, [40].log_data[9].valid := 1, [40].log_data[10].min := 1.0, [40].log_data[10].max := 1.0, [40].log_data[10].total := 3600.0, [40].log_data[10].time := 3600.0, [40].log_data[10].valid := 1, [40].log_data[11].time := 3600.0, [40].log_data[11].valid := 1, [40].log_data[12].min := 1.0, [40].log_data[12].max := 1.0,
        [40].log_data[12].total := 3600.0, [40].log_data[12].time := 3600.0, [40].log_data[12].valid := 1, [40].log_data[13].min := 1.0, [40].log_data[13].max := 1.0, [40].log_data[13].total := 3600.0, [40].log_data[13].time := 3600.0, [40].log_data[13].valid := 1, [40].log_data[14].time := 3600.0, [40].log_data[14].valid := 1, [40].log_data[15].time := 3600.0, [40].log_data[15].valid := 1, [40].log_data[16].time := 3600.0, [40].log_data[16].valid := 1, [40].log_data[17].min := 1.0, [40].log_data[17].max := 1.0, [40].log_data[17].total := 3600.0, [40].log_data[17].time := 3600.0, [40].log_data[17].valid := 1, [40].log_data[18].time := 3600.0, [40].log_data[18].valid := 1, [40].log_data[19].time := 3600.0, [40].log_data[19].valid := 1, [40].log_data[20].time := 3600.0, [40].log_data[20].valid := 1, [40].log_data[21].min := 1.0, [40].log_data[21].max := 1.0, [40].log_data[21].total := 3600.0, [40].log_data[21].time := 3600.0, [40].log_data[21].valid := 1, [40].log_data[22].time := 3600.0, [40].log_data[22].valid := 1, [40].log_data[23].time := 3600.0, [40].log_data[23].valid := 1, [40].log_data[24].time := 3600.0, [40].log_data[24].valid := 1, [40].log_data[25].time := 3600.0, [40].log_data[25].valid := 1, [40].log_data[26].time := 3600.0, [40].log_data[26].valid := 1, [40].log_data[27].time := 3600.0, [40].log_data[27].valid := 1, [40].log_data[28].time := 3600.0, [40].log_data[28].valid := 1, [40].log_data[29].min := 1.0, [40].log_data[29].max := 1.0, [40].log_data[29].total := 3600.0, [40].log_data[29].time := 3600.0, [40].log_data[29].valid := 1, [40].log_data[30].min := 1.0, [40].log_data[30].max := 1.0, [40].log_data[30].total := 3600.0, [40].log_data[30].time := 3600.0, [40].log_data[30].valid := 1, [40].log_data[31].max := 1.0, [40].log_data[31].total := 1440.7471, [40].log_data[31].time := 3600.0, [40].log_data[31].minminute := 3, [40].log_data[31].valid := 1, [40].log_data[32].max := 1.0,
        [40].log_data[32].total := 1629.998, [40].log_data[32].time := 3600.0, [40].log_data[32].maxminute := 5, [40].log_data[32].valid := 1, [40].log_data[33].time := 3600.0, [40].log_data[33].valid := 1, [40].log_data[34].time := 3600.0, [40].log_data[34].valid := 1, [40].log_data[35].max := 1.0, [40].log_data[35].total := 1558.2471, [40].log_data[35].time := 3600.0, [40].log_data[35].maxminute := 10, [40].log_data[35].valid := 1, [40].log_data[36].max := 1.0, [40].log_data[36].total := 1600.498, [40].log_data[36].time := 3600.0, [40].log_data[36].minminute := 8, [40].log_data[36].valid := 1, [40].log_data[37].max := 7.213641, [40].log_data[37].total := 3561.8157, [40].log_data[37].time := 3600.0, [40].log_data[37].maxminute := 38, [40].log_data[37].valid := 1, [40].log_data[38].time := 3600.0, [40].log_data[38].valid := 1, [40].log_data[39].min := 0.9956484, [40].log_data[39].max := 1.0214411, [40].log_data[39].total := 3620.6267, [40].log_data[39].time := 3600.0, [40].log_data[39].minminute := 44, [40].log_data[39].maxminute := 42, [40].log_data[39].valid := 1, [40].log_data[40].min := 7.561569, [40].log_data[40].max := 7.5934467, [40].log_data[40].total := 27291.11, [40].log_data[40].time := 3600.0, [40].log_data[40].minminute := 30, [40].log_data[40].maxminute := 49, [40].log_data[40].valid := 1, [40].log_data[41].min := 0.030980714, [40].log_data[41].max := 0.052769043, [40].log_data[41].total := 144.15436, [40].log_data[41].time := 3600.0, [40].log_data[41].minminute := 38, [40].log_data[41].maxminute := 19, [40].log_data[41].valid := 1, [40].log_data[42].min := 2.291996, [40].log_data[42].max := 2.2974136, [40].log_data[42].total := 8262.195, [40].log_data[42].time := 3600.0, [40].log_data[42].minminute := 31, [40].log_data[42].valid := 1, [40].log_data[43].min := -0.27999878, [40].log_data[43].max := -0.26000214, [40].log_data[43].total := -1007.8513, [40].log_data[43].time := 3600.0, [40].log_data[43].maxminute := 49, [40].log_data[43].valid := 1, [40].log_data[44].min := -0.3199997, [40].log_data[44].max := -0.30000305,
        [40].log_data[44].total := -1097.9509, [40].log_data[44].time := 3600.0, [40].log_data[44].valid := 1, [40].log_data[45].time := 3600.0, [40].log_data[45].valid := 1, [40].log_data[46].time := 3600.0, [40].log_data[46].valid := 1, [40].log_data[47].time := 3600.0, [40].log_data[47].valid := 1, [40].log_data[48].min := 6.632443, [40].log_data[48].max := 6.9069757, [40].log_data[48].total := 24330.906, [40].log_data[48].time := 3600.0, [40].log_data[48].minminute := 59, [40].log_data[48].maxminute := 45, [40].log_data[48].valid := 1, [40].log_data[49].min := 7.140262, [40].log_data[49].max := 9.621582, [40].log_data[49].total := 32295.566, [40].log_data[49].time := 3600.0, [40].log_data[49].minminute := 59, [40].log_data[49].maxminute := 38, [40].log_data[49].valid := 1, [40].log_data[50].min := 2.020996, [40].log_data[50].max := 2.1211047, [40].log_data[50].total := 7441.7427, [40].log_data[50].time := 3600.0, [40].log_data[50].minminute := 37, [40].log_data[50].maxminute := 47, [40].log_data[50].valid := 1, [40].log_data[51].time := 3600.0, [40].log_data[51].valid := 1, [40].log_data[52].min := -2.880005, [40].log_data[52].max := 0.11999512, [40].log_data[52].total := -7707.994, [40].log_data[52].time := 3600.0, [40].log_data[52].minminute := 5, [40].log_data[52].maxminute := 4, [40].log_data[52].valid := 1, [40].log_data[53].min := -2.7000046, [40].log_data[53].max := 0.22000122, [40].log_data[53].total := -7366.9062, [40].log_data[53].time := 3600.0, [40].log_data[53].minminute := 10, [40].log_data[53].maxminute := 41, [40].log_data[53].valid := 1, [40].log_data[54].max := 0.5315, [40].log_data[54].total := 1217.2075, [40].log_data[54].time := 3600.0, [40].log_data[54].minminute := 3, [40].log_data[54].maxminute := 5, [40].log_data[54].valid := 1, [40].log_data[55].max := 0.5385, [40].log_data[55].total := 1254.2375, [40].log_data[55].time := 3600.0, [40].log_data[55].minminute := 8, [40].log_data[55].maxminute := 10, [40].log_data[55].valid := 1, [40].log_data[56].min := 0.16020635, [40].log_data[56].max := 0.16063818,
        [40].log_data[56].total := 577.39026, [40].log_data[56].time := 3600.0, [40].log_data[56].minminute := 27, [40].log_data[56].valid := 1, [40].log_data[57].min := 0.28763872, [40].log_data[57].max := 0.2880313, [40].log_data[57].total := 1036.0773, [40].log_data[57].time := 3600.0, [40].log_data[57].minminute := 10, [40].log_data[57].maxminute := 3, [40].log_data[57].valid := 1, [40].log_data[58].time := 3600.0, [40].log_data[58].valid := 1, [40].log_data[59].time := 3600.0, [40].log_data[59].valid := 1, [40].log_data[60].valid := 1, [40].log_data[61].valid := 1, [40].log_data[62].valid := 1, [40].log_data[63].valid := 1, [40].log_data[64].valid := 1, [40].log_data[65].valid := 1, [40].log_data[66].valid := 1, [40].log_data[67].valid := 1, [40].log_data[68].valid := 1, [40].log_data[69].valid := 1, [40].log_data[70].valid := 1, [40].log_data[71].valid := 1, [40].log_data[72].valid := 1, [40].log_data[73].valid := 1, [40].log_data[74].valid := 1, [40].log_data[75].valid := 1, [40].log_data[76].valid := 1, [40].log_data[77].valid := 1, [40].log_data[78].valid := 1, [40].log_data[79].valid := 1, [40].log_data[80].valid := 1, [40].log_data[81].valid := 1, [40].log_data[82].valid := 1, [40].log_data[83].valid := 1, [40].log_data[84].valid := 1, [40].log_data[85].valid := 1, [40].log_data[86].valid := 1, [40].log_data[87].valid := 1, [40].log_data[88].valid := 1, [40].log_data[89].valid := 1, [40].log_data[90].valid := 1, [40].log_data[91].valid := 1, [40].log_data[92].valid := 1, [40].log_data[93].valid := 1, [40].log_data[94].valid := 1, [40].log_data[95].valid := 1, [40].log_data[96].valid := 1, [40].log_data[97].valid := 1, [40].log_data[98].valid := 1, [40].log_data[99].valid := 1, [40].log_data[100].valid := 1, [40].log_data[101].valid := 1, [40].log_data[102].valid := 1, [40].log_data[103].valid := 1, [40].log_data[104].valid := 1,
        [40].log_data[105].valid := 1, [40].log_data[106].valid := 1, [40].log_data[107].valid := 1, [40].log_data[108].valid := 1, [40].log_data[109].valid := 1, [40].log_data[110].valid := 1, [40].log_data[111].valid := 1, [40].log_data[112].valid := 1, [40].log_data[113].valid := 1, [40].log_data[114].valid := 1, [40].log_data[115].valid := 1, [40].log_data[116].valid := 1, [40].log_data[117].valid := 1, [40].log_data[118].valid := 1, [40].log_data[119].valid := 1, [40].log_data[120].valid := 1, [40].log_data[121].valid := 1, [40].log_data[122].valid := 1, [40].log_data[123].valid := 1, [40].log_data[124].valid := 1, [40].time.Year := 2023, [40].time.Month := 1, [40].time.Day := 14, [40].time.Hour := 19, [40].time.Minute := 59, [40].time.Second := 59, [41].log_data[0].min := 1.0, [41].log_data[0].max := 1.0, [41].log_data[0].total := 3600.0, [41].log_data[0].time := 3600.0, [41].log_data[0].valid := 1, [41].log_data[1].max := 1.0, [41].log_data[1].total := 245.749, [41].log_data[1].time := 3600.0, [41].log_data[1].maxminute := 55, [41].log_data[1].valid := 1, [41].log_data[2].max := 1.0, [41].log_data[2].total := 242.249, [41].log_data[2].time := 3600.0, [41].log_data[2].maxminute := 55, [41].log_data[2].valid := 1, [41].log_data[3].time := 3600.0, [41].log_data[3].valid := 1, [41].log_data[4].time := 3600.0, [41].log_data[4].valid := 1, [41].log_data[5].max := 1.0, [41].log_data[5].total := 125.5, [41].log_data[5].time := 3600.0, [41].log_data[5].maxminute := 57, [41].log_data[5].valid := 1, [41].log_data[6].time := 3600.0, [41].log_data[6].valid := 1, [41].log_data[7].time := 3600.0, [41].log_data[7].valid := 1, [41].log_data[8].min := 1.0, [41].log_data[8].max := 1.0, [41].log_data[8].total := 3600.0, [41].log_data[8].time := 3600.0, [41].log_data[8].valid := 1, [41].log_data[9].min := 1.0,
        [41].log_data[9].max := 1.0, [41].log_data[9].total := 3600.0, [41].log_data[9].time := 3600.0, [41].log_data[9].valid := 1, [41].log_data[10].min := 1.0, [41].log_data[10].max := 1.0, [41].log_data[10].total := 3600.0, [41].log_data[10].time := 3600.0, [41].log_data[10].valid := 1, [41].log_data[11].time := 3600.0, [41].log_data[11].valid := 1, [41].log_data[12].min := 1.0, [41].log_data[12].max := 1.0, [41].log_data[12].total := 3600.0, [41].log_data[12].time := 3600.0, [41].log_data[12].valid := 1, [41].log_data[13].min := 1.0, [41].log_data[13].max := 1.0, [41].log_data[13].total := 3600.0, [41].log_data[13].time := 3600.0, [41].log_data[13].valid := 1, [41].log_data[14].time := 3600.0, [41].log_data[14].valid := 1, [41].log_data[15].time := 3600.0, [41].log_data[15].valid := 1, [41].log_data[16].time := 3600.0, [41].log_data[16].valid := 1, [41].log_data[17].min := 1.0, [41].log_data[17].max := 1.0, [41].log_data[17].total := 3600.0, [41].log_data[17].time := 3600.0, [41].log_data[17].valid := 1, [41].log_data[18].time := 3600.0, [41].log_data[18].valid := 1, [41].log_data[19].time := 3600.0, [41].log_data[19].valid := 1, [41].log_data[20].time := 3600.0, [41].log_data[20].valid := 1, [41].log_data[21].min := 1.0, [41].log_data[21].max := 1.0, [41].log_data[21].total := 3600.0, [41].log_data[21].time := 3600.0, [41].log_data[21].valid := 1, [41].log_data[22].time := 3600.0, [41].log_data[22].valid := 1, [41].log_data[23].time := 3600.0, [41].log_data[23].valid := 1, [41].log_data[24].time := 3600.0, [41].log_data[24].valid := 1, [41].log_data[25].time := 3600.0, [41].log_data[25].valid := 1, [41].log_data[26].time := 3600.0, [41].log_data[26].valid := 1, [41].log_data[27].time := 3600.0, [41].log_data[27].valid := 1, [41].log_data[28].time := 3600.0, [41].log_data[28].valid := 1, [41].log_data[29].min := 1.0, [41].log_data[29].max := 1.0, [41].log_data[29].total := 3600.0,
        [41].log_data[29].time := 3600.0, [41].log_data[29].valid := 1, [41].log_data[30].min := 1.0, [41].log_data[30].max := 1.0, [41].log_data[30].total := 3600.0, [41].log_data[30].time := 3600.0, [41].log_data[30].valid := 1, [41].log_data[31].max := 1.0, [41].log_data[31].total := 1491.498, [41].log_data[31].time := 3600.0, [41].log_data[31].minminute := 6, [41].log_data[31].valid := 1, [41].log_data[32].max := 1.0, [41].log_data[32].total := 1629.7471, [41].log_data[32].time := 3600.0, [41].log_data[32].maxminute := 8, [41].log_data[32].valid := 1, [41].log_data[33].time := 3600.0, [41].log_data[33].valid := 1, [41].log_data[34].time := 3600.0, [41].log_data[34].valid := 1, [41].log_data[35].max := 1.0, [41].log_data[35].total := 1440.7471, [41].log_data[35].time := 3600.0, [41].log_data[35].minminute := 1, [41].log_data[35].valid := 1, [41].log_data[36].max := 1.0, [41].log_data[36].total := 1629.7471, [41].log_data[36].time := 3600.0, [41].log_data[36].maxminute := 2, [41].log_data[36].valid := 1, [41].log_data[37].max := 7.508471, [41].log_data[37].total := 1814.5615, [41].log_data[37].time := 3600.0, [41].log_data[37].maxminute := 57, [41].log_data[37].valid := 1, [41].log_data[38].time := 3600.0, [41].log_data[38].valid := 1, [41].log_data[39].min := 0.9994172, [41].log_data[39].max := 1.0225011, [41].log_data[39].total := 3630.756, [41].log_data[39].time := 3600.0, [41].log_data[39].minminute := 59, [41].log_data[39].maxminute := 57, [41].log_data[39].valid := 1, [41].log_data[40].min := 7.5629425, [41].log_data[40].max := 7.597843, [41].log_data[40].total := 27299.383, [41].log_data[40].time := 3600.0, [41].log_data[40].minminute := 43, [41].log_data[40].maxminute := 24, [41].log_data[40].valid := 1, [41].log_data[41].min := 0.032943603, [41].log_data[41].max := 0.04766553, [41].log_data[41].total := 140.96608, [41].log_data[41].time := 3600.0, [41].log_data[41].minminute := 1, [41].log_data[41].maxminute := 41, [41].log_data[41].valid := 1, [41].log_data[42].min := 2.292467,
        [41].log_data[42].max := 2.2970603, [41].log_data[42].total := 8262.012, [41].log_data[42].time := 3600.0, [41].log_data[42].minminute := 36, [41].log_data[42].maxminute := 59, [41].log_data[42].valid := 1, [41].log_data[43].min := -0.27999878, [41].log_data[43].max := -0.26000214, [41].log_data[43].total := -1007.55273, [41].log_data[43].time := 3600.0, [41].log_data[43].maxminute := 5, [41].log_data[43].valid := 1, [41].log_data[44].min := -0.3199997, [41].log_data[44].max := -0.30000305, [41].log_data[44].total := -1083.7208, [41].log_data[44].time := 3600.0, [41].log_data[44].valid := 1, [41].log_data[45].time := 3600.0, [41].log_data[45].valid := 1, [41].log_data[46].time := 3600.0, [41].log_data[46].valid := 1, [41].log_data[47].time := 3600.0, [41].log_data[47].valid := 1, [41].log_data[48].min := 6.5824285, [41].log_data[48].max := 6.9366555, [41].log_data[48].total := 24229.58, [41].log_data[48].time := 3600.0, [41].log_data[48].minminute := 6, [41].log_data[48].maxminute := 59, [41].log_data[48].valid := 1, [41].log_data[49].min := 7.0688124, [41].log_data[49].max := 9.622562, [41].log_data[49].total := 31563.205, [41].log_data[49].time := 3600.0, [41].log_data[49].minminute := 2, [41].log_data[49].maxminute := 56, [41].log_data[49].valid := 1, [41].log_data[50].min := 2.0179338, [41].log_data[50].max := 2.1060295, [41].log_data[50].total := 7430.741, [41].log_data[50].time := 3600.0, [41].log_data[50].minminute := 57, [41].log_data[50].valid := 1, [41].log_data[51].time := 3600.0, [41].log_data[51].valid := 1, [41].log_data[52].min := -2.7600021, [41].log_data[52].max := 0.11999512, [41].log_data[52].total := -7808.743, [41].log_data[52].time := 3600.0, [41].log_data[52].minminute := 8, [41].log_data[52].maxminute := 6, [41].log_data[52].valid := 1, [41].log_data[53].min := -2.5, [41].log_data[53].max := 0.27999878, [41].log_data[53].total := -7146.68, [41].log_data[53].time := 3600.0, [41].log_data[53].minminute := 38, [41].log_data[53].maxminute := 12, [41].log_data[53].valid := 1, [41].log_data[54].max := 0.5325,
        [41].log_data[54].total := 1239.4784, [41].log_data[54].time := 3600.0, [41].log_data[54].minminute := 6, [41].log_data[54].maxminute := 8, [41].log_data[54].valid := 1, [41].log_data[55].max := 0.519, [41].log_data[55].total := 1217.3094, [41].log_data[55].time := 3600.0, [41].log_data[55].minminute := 1, [41].log_data[55].maxminute := 2, [41].log_data[55].valid := 1, [41].log_data[56].min := 0.16024561, [41].log_data[56].max := 0.16067745, [41].log_data[56].total := 577.4652, [41].log_data[56].time := 3600.0, [41].log_data[56].maxminute := 24, [41].log_data[56].valid := 1, [41].log_data[57].min := 0.2861862, [41].log_data[57].max := 0.28795278, [41].log_data[57].total := 1031.6627, [41].log_data[57].time := 3600.0, [41].log_data[57].minminute := 17, [41].log_data[57].valid := 1, [41].log_data[58].time := 3600.0, [41].log_data[58].valid := 1, [41].log_data[59].time := 3600.0, [41].log_data[59].valid := 1, [41].log_data[60].valid := 1, [41].log_data[61].valid := 1, [41].log_data[62].valid := 1, [41].log_data[63].valid := 1, [41].log_data[64].valid := 1, [41].log_data[65].valid := 1, [41].log_data[66].valid := 1, [41].log_data[67].valid := 1, [41].log_data[68].valid := 1, [41].log_data[69].valid := 1, [41].log_data[70].valid := 1, [41].log_data[71].valid := 1, [41].log_data[72].valid := 1, [41].log_data[73].valid := 1, [41].log_data[74].valid := 1, [41].log_data[75].valid := 1, [41].log_data[76].valid := 1, [41].log_data[77].valid := 1, [41].log_data[78].valid := 1, [41].log_data[79].valid := 1, [41].log_data[80].valid := 1, [41].log_data[81].valid := 1, [41].log_data[82].valid := 1, [41].log_data[83].valid := 1, [41].log_data[84].valid := 1, [41].log_data[85].valid := 1, [41].log_data[86].valid := 1, [41].log_data[87].valid := 1, [41].log_data[88].valid := 1, [41].log_data[89].valid := 1, [41].log_data[90].valid := 1, [41].log_data[91].valid := 1, [41].log_data[92].valid := 1,
        [41].log_data[93].valid := 1, [41].log_data[94].valid := 1, [41].log_data[95].valid := 1, [41].log_data[96].valid := 1, [41].log_data[97].valid := 1, [41].log_data[98].valid := 1, [41].log_data[99].valid := 1, [41].log_data[100].valid := 1, [41].log_data[101].valid := 1, [41].log_data[102].valid := 1, [41].log_data[103].valid := 1, [41].log_data[104].valid := 1, [41].log_data[105].valid := 1, [41].log_data[106].valid := 1, [41].log_data[107].valid := 1, [41].log_data[108].valid := 1, [41].log_data[109].valid := 1, [41].log_data[110].valid := 1, [41].log_data[111].valid := 1, [41].log_data[112].valid := 1, [41].log_data[113].valid := 1, [41].log_data[114].valid := 1, [41].log_data[115].valid := 1, [41].log_data[116].valid := 1, [41].log_data[117].valid := 1, [41].log_data[118].valid := 1, [41].log_data[119].valid := 1, [41].log_data[120].valid := 1, [41].log_data[121].valid := 1, [41].log_data[122].valid := 1, [41].log_data[123].valid := 1, [41].log_data[124].valid := 1, [41].time.Year := 2023, [41].time.Month := 1, [41].time.Day := 14, [41].time.Hour := 20, [41].time.Minute := 59, [41].time.Second := 59, [42].log_data[0].min := 1.0, [42].log_data[0].max := 1.0, [42].log_data[0].total := 3600.0, [42].log_data[0].time := 3600.0, [42].log_data[0].valid := 1, [42].log_data[1].max := 1.0, [42].log_data[1].total := 303.751, [42].log_data[1].time := 3600.0, [42].log_data[1].minminute := 5, [42].log_data[1].valid := 1, [42].log_data[2].max := 1.0, [42].log_data[2].total := 303.751, [42].log_data[2].time := 3600.0, [42].log_data[2].minminute := 5, [42].log_data[2].valid := 1, [42].log_data[3].time := 3600.0, [42].log_data[3].valid := 1, [42].log_data[4].time := 3600.0, [42].log_data[4].valid := 1, [42].log_data[5].max := 1.0, [42].log_data[5].total := 105.5, [42].log_data[5].time := 3600.0,
        [42].log_data[5].maxminute := 1, [42].log_data[5].valid := 1, [42].log_data[6].time := 3600.0, [42].log_data[6].valid := 1, [42].log_data[7].time := 3600.0, [42].log_data[7].valid := 1, [42].log_data[8].min := 1.0, [42].log_data[8].max := 1.0, [42].log_data[8].total := 3600.0, [42].log_data[8].time := 3600.0, [42].log_data[8].valid := 1, [42].log_data[9].min := 1.0, [42].log_data[9].max := 1.0, [42].log_data[9].total := 3600.0, [42].log_data[9].time := 3600.0, [42].log_data[9].valid := 1, [42].log_data[10].min := 1.0, [42].log_data[10].max := 1.0, [42].log_data[10].total := 3600.0, [42].log_data[10].time := 3600.0, [42].log_data[10].valid := 1, [42].log_data[11].time := 3600.0, [42].log_data[11].valid := 1, [42].log_data[12].min := 1.0, [42].log_data[12].max := 1.0, [42].log_data[12].total := 3600.0, [42].log_data[12].time := 3600.0, [42].log_data[12].valid := 1, [42].log_data[13].min := 1.0, [42].log_data[13].max := 1.0, [42].log_data[13].total := 3600.0, [42].log_data[13].time := 3600.0, [42].log_data[13].valid := 1, [42].log_data[14].time := 3600.0, [42].log_data[14].valid := 1, [42].log_data[15].time := 3600.0, [42].log_data[15].valid := 1, [42].log_data[16].time := 3600.0, [42].log_data[16].valid := 1, [42].log_data[17].min := 1.0, [42].log_data[17].max := 1.0, [42].log_data[17].total := 3600.0, [42].log_data[17].time := 3600.0, [42].log_data[17].valid := 1, [42].log_data[18].time := 3600.0, [42].log_data[18].valid := 1, [42].log_data[19].time := 3600.0, [42].log_data[19].valid := 1, [42].log_data[20].time := 3600.0, [42].log_data[20].valid := 1, [42].log_data[21].min := 1.0, [42].log_data[21].max := 1.0, [42].log_data[21].total := 3600.0, [42].log_data[21].time := 3600.0, [42].log_data[21].valid := 1, [42].log_data[22].time := 3600.0, [42].log_data[22].valid := 1, [42].log_data[23].time := 3600.0, [42].log_data[23].valid := 1, [42].log_data[24].time := 3600.0,
        [42].log_data[24].valid := 1, [42].log_data[25].time := 3600.0, [42].log_data[25].valid := 1, [42].log_data[26].time := 3600.0, [42].log_data[26].valid := 1, [42].log_data[27].time := 3600.0, [42].log_data[27].valid := 1, [42].log_data[28].time := 3600.0, [42].log_data[28].valid := 1, [42].log_data[29].min := 1.0, [42].log_data[29].max := 1.0, [42].log_data[29].total := 3600.0, [42].log_data[29].time := 3600.0, [42].log_data[29].valid := 1, [42].log_data[30].min := 1.0, [42].log_data[30].max := 1.0, [42].log_data[30].total := 3600.0, [42].log_data[30].time := 3600.0, [42].log_data[30].valid := 1, [42].log_data[31].max := 1.0, [42].log_data[31].total := 1629.7471, [42].log_data[31].time := 3600.0, [42].log_data[31].valid := 1, [42].log_data[32].max := 1.0, [42].log_data[32].total := 1478.2471, [42].log_data[32].time := 3600.0, [42].log_data[32].maxminute := 11, [42].log_data[32].valid := 1, [42].log_data[33].time := 3600.0, [42].log_data[33].valid := 1, [42].log_data[34].time := 3600.0, [42].log_data[34].valid := 1, [42].log_data[35].max := 1.0, [42].log_data[35].total := 1440.498, [42].log_data[35].time := 3600.0, [42].log_data[35].minminute := 4, [42].log_data[35].valid := 1, [42].log_data[36].max := 1.0, [42].log_data[36].total := 1629.7471, [42].log_data[36].time := 3600.0, [42].log_data[36].maxminute := 5, [42].log_data[36].valid := 1, [42].log_data[37].max := 7.410718, [42].log_data[37].total := 1768.5547, [42].log_data[37].time := 3600.0, [42].log_data[37].minminute := 4, [42].log_data[37].valid := 1, [42].log_data[38].time := 3600.0, [42].log_data[38].valid := 1, [42].log_data[39].min := 0.99882835, [42].log_data[39].max := 1.0201455, [42].log_data[39].total := 3638.6985, [42].log_data[39].time := 3600.0, [42].log_data[39].minminute := 3, [42].log_data[39].maxminute := 1, [42].log_data[39].valid := 1, [42].log_data[40].min := 7.557446, [42].log_data[40].max := 7.5989423, [42].log_data[40].total := 27304.922, [42].log_data[40].time := 3600.0,
